  MoveL 6541 to (12.86, -64.22, -148.97) mm, rotated rx 81.04 ry 30.21 rz 20.91 deg; joints [-5.811, -13.888, 75.553, 102.149, 106.889, 54.392, -153.967]
  MoveL 6542 to (13.22, -64.48, -148.9) mm, rotated rx 81.04 ry 30.21 rz 20.91 deg; joints [-5.821, -13.905, 75.562, 102.142, 106.892, 54.402, -153.967]
  MoveL 6543 to (13.58, -64.78, -148.85) mm, rotated rx 81.04 ry 30.21 rz 20.91 deg; joints [-5.832, -13.921, 75.565, 102.137, 106.894, 54.415, -153.967]
  MoveL 6544 to (13.94, -65.11, -148.82) mm, rotated rx 81.04 ry 30.21 rz 20.91 deg; joints [-5.843, -13.936, 75.566, 102.132, 106.896, 54.431, -153.967]
  MoveL 6545 to (14.32, -65.47, -148.8) mm, rotated rx 81.04 ry 30.21 rz 20.91 deg; joints [-5.855, -13.951, 75.564, 102.127, 106.898, 54.45, -153.967]
  MoveL 6546 to (14.69, -65.84, -148.8) mm, rotated rx 81.04 ry 30.21 rz 20.91 deg; joints [-5.866, -13.965, 75.559, 102.123, 106.9, 54.47, -153.967]
  MoveL 6547 to (15.03, -66.17, -148.79) mm, rotated rx 81.04 ry 30.21 rz 20.91 deg; joints [-5.876, -13.978, 75.556, 102.118, 106.901, 54.487, -153.967]
  MoveL 6548 to (15.34, -66.45, -148.76) mm, rotated rx 81.04 ry 30.21 rz 20.91 deg; joints [-5.886, -13.991, 75.556, 102.114, 106.903, 54.501, -153.967]
  MoveL 6549 to (15.69, -66.78, -148.75) mm, rotated rx 81.04 ry 30.21 rz 20.91 deg; joints [-5.897, -14.004, 75.554, 102.11, 106.904, 54.519, -153.967]
  MoveL 6550 to (16.06, -67.16, -148.75) mm, rotated rx 81.04 ry 30.21 rz 20.91 deg; joints [-5.908, -14.018, 75.549, 102.106, 106.906, 54.539, -153.967]
  MoveL 6551 to (16.5, -67.58, -148.73) mm, rotated rx 81.04 ry 30.21 rz 20.91 deg; joints [-5.922, -14.035, 75.546, 102.1, 106.908, 54.561, -153.967]
  MoveL 6552 to (17, -68.06, -148.69) mm, rotated rx 81.04 ry 30.21 rz 20.91 deg; joints [-5.937, -14.056, 75.545, 102.094, 106.91, 54.585, -153.967]
  MoveL 6553 to (17.44, -68.48, -148.67) mm, rotated rx 81.04 ry 30.21 rz 20.91 deg; joints [-5.95, -14.074, 75.542, 102.089, 106.912, 54.607, -153.967]
  MoveL 6554 to (17.9, -68.93, -148.64) mm, rotated rx 81.04 ry 30.21 rz 20.91 deg; joints [-5.964, -14.092, 75.54, 102.083, 106.915, 54.63, -153.967]
  MoveL 6555 to (18.43, -69.41, -148.6) mm, rotated rx 81.04 ry 30.21 rz 20.91 deg; joints [-5.98, -14.113, 75.539, 102.076, 106.917, 54.654, -153.967]
  MoveL 6556 to (18.85, -69.82, -148.59) mm, rotated rx 81.04 ry 30.21 rz 20.91 deg; joints [-5.993, -14.13, 75.535, 102.071, 106.919, 54.676, -153.967]
  MoveL 6557 to (19.24, -70.21, -148.59) mm, rotated rx 81.04 ry 30.21 rz 20.91 deg; joints [-6.005, -14.144, 75.53, 102.066, 106.921, 54.697, -153.967]
  MoveL 6558 to (20.34, -71.32, -148.59) mm, rotated rx 81.04 ry 30.21 rz 20.91 deg; joints [-6.04, -14.184, 75.514, 102.054, 106.925, 54.758, -153.967]
  MoveL 6559 to (21.31, -72.4, -148.67) mm, rotated rx 81.04 ry 30.21 rz 20.91 deg; joints [-6.071, -14.215, 75.486, 102.045, 106.928, 54.822, -153.967]
  MoveL 6560 to (21.99, -73.38, -148.93) mm, rotated rx 81.04 ry 30.21 rz 20.91 deg; joints [-6.094, -14.226, 75.434, 102.044, 106.925, 54.889, -153.967]
  MoveL 6561 to (22.38, -74.25, -149.35) mm, rotated rx 81.04 ry 30.21 rz 20.91 deg; joints [-6.11, -14.216, 75.357, 102.051, 106.919, 54.959, -153.967]
  MoveL 6562 to (22.46, -74.65, -149.62) mm, rotated rx 81.04 ry 30.21 rz 20.91 deg; joints [-6.116, -14.204, 75.309, 102.057, 106.914, 54.996, -153.967]
  MoveL 6563 to (22.47, -75.03, -149.94) mm, rotated rx 81.04 ry 30.21 rz 20.91 deg; joints [-6.119, -14.187, 75.256, 102.064, 106.908, 55.033, -153.967]
  MoveL 6564 to (22.26, -75.71, -150.7) mm, rotated rx 81.04 ry 30.21 rz 20.91 deg; joints [-6.121, -14.137, 75.131, 102.086, 106.893, 55.111, -153.967]
  MoveL 6565 to (21.77, -76.28, -151.62) mm, rotated rx 81.04 ry 30.21 rz 20.91 deg; joints [-6.115, -14.068, 74.981, 102.115, 106.873, 55.192, -153.967]
  MoveL 6566 to (19.9, -77.13, -153.99) mm, rotated rx 81.04 ry 30.21 rz 20.91 deg; joints [-6.08, -13.868, 74.607, 102.195, 106.821, 55.366, -153.967]
  MoveL 6567 to (17.5, -77.39, -156.35) mm, rotated rx 81.04 ry 30.21 rz 20.91 deg; joints [-6.031, -13.647, 74.243, 102.279, 106.766, 55.507, -153.967]
  MoveL 6568 to (15.25, -76.85, -158.04) mm, rotated rx 81.04 ry 30.21 rz 20.91 deg; joints [-5.978, -13.467, 73.999, 102.342, 106.727, 55.567, -153.967]
  MoveL 6569 to (14.17, -76.28, -158.63) mm, rotated rx 81.04 ry 30.21 rz 20.91 deg; joints [-5.951, -13.393, 73.921, 102.365, 106.714, 55.567, -153.967]
  MoveL 6570 to (13.12, -75.52, -159.05) mm, rotated rx 81.04 ry 30.21 rz 20.91 deg; joints [-5.923, -13.329, 73.874, 102.384, 106.704, 55.546, -153.967]
  MoveL 6571 to (11.13, -73.39, -159.39) mm, rotated rx 81.04 ry 30.21 rz 20.91 deg; joints [-5.865, -13.232, 73.871, 102.405, 106.696, 55.444, -153.967]
  MoveL 6572 to (8.58, -70.06, -159.39) mm, rotated rx 81.04 ry 30.21 rz 20.91 deg; joints [-5.787, -13.13, 73.945, 102.419, 106.697, 55.257, -153.967]
  MoveL 6573 to (8.24, -69.63, -159.41) mm, rotated rx 81.04 ry 30.21 rz 20.91 deg; joints [-5.777, -13.115, 73.952, 102.421, 106.697, 55.234, -153.967]
  MoveL 6574 to (7.9, -69.23, -159.45) mm, rotated rx 81.04 ry 30.21 rz 20.91 deg; joints [-5.767, -13.099, 73.955, 102.424, 106.696, 55.213, -153.967]
  MoveL 6575 to (7.54, -68.84, -159.51) mm, rotated rx 81.04 ry 30.21 rz 20.91 deg; joints [-5.757, -13.082, 73.955, 102.428, 106.695, 55.194, -153.967]
  MoveL 6576 to (7.18, -68.47, -159.59) mm, rotated rx 81.04 ry 30.21 rz 20.91 deg; joints [-5.746, -13.062, 73.951, 102.432, 106.693, 55.178, -153.967]
  MoveL 6577 to (6.83, -68.1, -159.67) mm, rotated rx 81.04 ry 30.21 rz 20.91 deg; joints [-5.736, -13.044, 73.947, 102.436, 106.692, 55.161, -153.967]
  MoveL 6578 to (6.52, -67.73, -159.71) mm, rotated rx 81.04 ry 30.21 rz 20.91 deg; joints [-5.727, -13.029, 73.95, 102.439, 106.691, 55.143, -153.967]
  MoveL 6579 to (6.21, -67.35, -159.72) mm, rotated rx 81.04 ry 30.21 rz 20.91 deg; joints [-5.718, -13.016, 73.956, 102.441, 106.691, 55.122, -153.967]
  MoveL 6580 to (5.9, -66.94, -159.72) mm, rotated rx 81.04 ry 30.21 rz 20.91 deg; joints [-5.708, -13.003, 73.965, 102.443, 106.691, 55.099, -153.967]
  MoveL 6581 to (5.5, -66.45, -159.76) mm, rotated rx 81.04 ry 30.21 rz 20.91 deg; joints [-5.697, -12.985, 73.97, 102.446, 106.69, 55.074, -153.967]
  MoveL 6582 to (5.06, -65.93, -159.82) mm, rotated rx 81.04 ry 30.21 rz 20.91 deg; joints [-5.683, -12.964, 73.973, 102.45, 106.689, 55.048, -153.967]
  MoveL 6583 to (4.66, -65.49, -159.84) mm, rotated rx 81.04 ry 30.21 rz 20.91 deg; joints [-5.672, -12.948, 73.979, 102.453, 106.688, 55.024, -153.967]
  MoveL 6584 to (4.27, -65.09, -159.85) mm, rotated rx 81.04 ry 30.21 rz 20.91 deg; joints [-5.659, -12.932, 73.982, 102.458, 106.687, 55.004, -153.967]
  MoveL 6585 to (3.84, -64.74, -159.85) mm, rotated rx 81.04 ry 30.21 rz 20.91 deg; joints [-5.646, -12.917, 73.983, 102.464, 106.684, 54.986, -153.967]
  MoveL 6586 to (3.33, -64.47, -159.85) mm, rotated rx 81.04 ry 30.21 rz 20.91 deg; joints [-5.63, -12.901, 73.977, 102.475, 106.679, 54.974, -153.967]
  MoveL 6587 to (2.76, -64.25, -159.85) mm, rotated rx 81.04 ry 30.21 rz 20.91 deg; joints [-5.612, -12.885, 73.967, 102.488, 106.672, 54.966, -153.967]
  MoveL 6588 to (4.06, -65.14, -160.81) mm, rotated rx 81.04 ry 30.21 rz 20.91 deg; joints [-5.664, -12.861, 73.865, 102.468, 106.679, 55.051, -153.967]
  MoveL 6589 to (2.83, -64.96, -161.23) mm, rotated rx 81.04 ry 30.21 rz 20.91 deg; joints [-5.63, -12.798, 73.778, 102.504, 106.658, 55.071, -153.967]
  MoveL 6590 to (1.45, -64.66, -161.56) mm, rotated rx 81.04 ry 30.21 rz 20.91 deg; joints [-5.59, -12.737, 73.704, 102.541, 106.636, 55.081, -153.967]
  MoveL 6591 to (-0.1, -64.24, -161.81) mm, rotated rx 81.04 ry 30.21 rz 20.91 deg; joints [-5.544, -12.676, 73.637, 102.582, 106.613, 55.081, -153.967]
  MoveL 6592 to (-2.13, -63.57, -161.92) mm, rotated rx 81.04 ry 30.21 rz 20.91 deg; joints [-5.481, -12.609, 73.579, 102.632, 106.585, 55.065, -153.967]
  MoveL 6593 to (-4.16, -62.93, -162.15) mm, rotated rx 81.04 ry 30.21 rz 20.91 deg; joints [-5.42, -12.534, 73.506, 102.683, 106.557, 55.056, -153.967]
  MoveL 6594 to (-6.19, -62.26, -162.26) mm, rotated rx 81.04 ry 30.21 rz 20.91 deg; joints [-5.358, -12.467, 73.447, 102.733, 106.529, 55.041, -153.967]
  MoveL 6595 to (-8.21, -61.59, -162.38) mm, rotated rx 81.04 ry 30.21 rz 20.91 deg; joints [-5.295, -12.399, 73.388, 102.783, 106.501, 55.025, -153.967]
  MoveL 6596 to (-10.24, -60.93, -162.61) mm, rotated rx 81.04 ry 30.21 rz 20.91 deg; joints [-5.234, -12.323, 73.315, 102.834, 106.473, 55.016, -153.967]
  MoveL 6597 to (-12.26, -60.25, -162.73) mm, rotated rx 81.04 ry 30.21 rz 20.91 deg; joints [-5.172, -12.255, 73.255, 102.884, 106.445, 55.001, -153.967]
  MoveL 6598 to (-14.28, -59.57, -162.85) mm, rotated rx 81.04 ry 30.21 rz 20.91 deg; joints [-5.11, -12.187, 73.194, 102.934, 106.418, 54.986, -153.967]
  MoveL 6599 to (-16.62, -58.79, -163.01) mm, rotated rx 81.04 ry 30.21 rz 20.91 deg; joints [-5.038, -12.107, 73.122, 102.992, 106.386, 54.97, -153.967]
  MoveL 6600 to (-18.61, -58.12, -163.21) mm, rotated rx 81.04 ry 30.21 rz 20.91 deg; joints [-4.978, -12.034, 73.054, 103.041, 106.358, 54.958, -153.967]
  MoveL 6601 to (-20.79, -57.37, -163.41) mm, rotated rx 81.04 ry 30.21 rz 20.91 deg; joints [-4.912, -11.955, 72.98, 103.096, 106.328, 54.945, -153.967]
  MoveL 6602 to (-22.93, -56.64, -163.66) mm, rotated rx 81.04 ry 30.21 rz 20.91 deg; joints [-4.848, -11.873, 72.901, 103.149, 106.299, 54.935, -153.967]
  MoveL 6603 to (-24.95, -55.95, -163.78) mm, rotated rx 81.04 ry 30.21 rz 20.91 deg; joints [-4.786, -11.804, 72.839, 103.199, 106.271, 54.92, -153.967]
  MoveL 6604 to (-26.97, -55.26, -163.78) mm, rotated rx 81.04 ry 30.21 rz 20.91 deg; joints [-4.722, -11.743, 72.791, 103.249, 106.244, 54.9, -153.967]
  MoveL 6605 to (-28.96, -54.57, -163.86) mm, rotated rx 81.04 ry 30.21 rz 20.91 deg; joints [-4.661, -11.678, 72.735, 103.298, 106.217, 54.884, -153.967]
  MoveL 6606 to (-30.9, -53.88, -164.07) mm, rotated rx 81.04 ry 30.21 rz 20.91 deg; joints [-4.602, -11.604, 72.665, 103.346, 106.191, 54.873, -153.967]
  MoveL 6607 to (-33.06, -53.09, -164.42) mm, rotated rx 81.04 ry 30.21 rz 20.91 deg; joints [-4.539, -11.513, 72.574, 103.4, 106.161, 54.866, -153.967]
  MoveL 6608 to (-34.75, -52.47, -164.63) mm, rotated rx 81.04 ry 30.21 rz 20.91 deg; joints [-4.488, -11.446, 72.51, 103.442, 106.137, 54.857, -153.967]
  MoveL 6609 to (-37.05, -51.6, -164.93) mm, rotated rx 81.04 ry 30.21 rz 20.91 deg; joints [-4.419, -11.354, 72.423, 103.498, 106.106, 54.844, -153.967]
  MoveL 6610 to (-39.13, -50.86, -165.03) mm, rotated rx 81.04 ry 30.21 rz 20.91 deg; joints [-4.355, -11.283, 72.361, 103.55, 106.078, 54.828, -153.967]
  MoveL 6611 to (-41.15, -50.17, -165.05) mm, rotated rx 81.04 ry 30.21 rz 20.91 deg; joints [-4.292, -11.221, 72.308, 103.6, 106.051, 54.81, -153.967]
  MoveL 6612 to (-41.68, -49.46, -165.84) mm, rotated rx 81.04 ry 30.21 rz 20.91 deg; joints [-4.285, -11.142, 72.231, 103.606, 106.048, 54.808, -153.967]
  MoveL 6613 to (-41.25, -49.43, -166.23) mm, rotated rx 81.04 ry 30.21 rz 20.91 deg; joints [-4.303, -11.126, 72.207, 103.593, 106.054, 54.818, -153.967]
  MoveL 6614 to (-41.11, -49.43, -166.47) mm, rotated rx 81.04 ry 30.21 rz 20.91 deg; joints [-4.31, -11.113, 72.185, 103.589, 106.056, 54.828, -153.967]
  MoveL 6615 to (-41.24, -49.46, -166.6) mm, rotated rx 81.04 ry 30.21 rz 20.91 deg; joints [-4.307, -11.101, 72.163, 103.594, 106.052, 54.837, -153.967]
  MoveL 6616 to (-41.63, -49.55, -166.62) mm, rotated rx 81.04 ry 30.21 rz 20.91 deg; joints [-4.296, -11.09, 72.139, 103.608, 106.044, 54.849, -153.967]
  MoveL 6617 to (-42.08, -49.66, -166.63) mm, rotated rx 81.04 ry 30.21 rz 20.91 deg; joints [-4.281, -11.079, 72.114, 103.624, 106.033, 54.862, -153.967]
  MoveL 6618 to (-43.6, -50.07, -166.63) mm, rotated rx 81.04 ry 30.21 rz 20.91 deg; joints [-4.234, -11.043, 72.028, 103.678, 105.999, 54.907, -153.967]
  MoveL 6619 to (-44.14, -50.2, -166.65) mm, rotated rx 81.04 ry 30.21 rz 20.91 deg; joints [-4.217, -11.029, 71.996, 103.697, 105.987, 54.923, -153.967]
  MoveL 6620 to (-44.68, -50.31, -166.69) mm, rotated rx 81.04 ry 30.21 rz 20.91 deg; joints [-4.201, -11.013, 71.962, 103.716, 105.975, 54.939, -153.967]
  MoveL 6621 to (-45.24, -50.41, -166.77) mm, rotated rx 81.04 ry 30.21 rz 20.91 deg; joints [-4.184, -10.993, 71.923, 103.735, 105.963, 54.956, -153.967]
  MoveL 6622 to (-45.79, -50.51, -166.83) mm, rotated rx 81.04 ry 30.21 rz 20.91 deg; joints [-4.168, -10.976, 71.888, 103.754, 105.951, 54.972, -153.967]
  MoveL 6623 to (-46.3, -50.63, -166.86) mm, rotated rx 81.04 ry 30.21 rz 20.91 deg; joints [-4.152, -10.961, 71.857, 103.772, 105.939, 54.987, -153.967]
  MoveL 6624 to (-46.79, -50.75, -166.88) mm, rotated rx 81.04 ry 30.21 rz 20.91 deg; joints [-4.137, -10.949, 71.828, 103.789, 105.928, 55.002, -153.967]
  MoveL 6625 to (-47.24, -50.84, -166.92) mm, rotated rx 81.04 ry 30.21 rz 20.91 deg; joints [-4.123, -10.934, 71.799, 103.804, 105.918, 55.015, -153.967]
  MoveL 6626 to (-47.67, -50.93, -166.96) mm, rotated rx 81.04 ry 30.21 rz 20.91 deg; joints [-4.11, -10.921, 71.771, 103.819, 105.909, 55.028, -153.967]
  MoveL 6627 to (-48.15, -51.04, -166.98) mm, rotated rx 81.04 ry 30.21 rz 20.91 deg; joints [-4.095, -10.908, 71.743, 103.836, 105.898, 55.042, -153.967]
  MoveL 6628 to (-48.72, -51.18, -167) mm, rotated rx 81.04 ry 30.21 rz 20.91 deg; joints [-4.077, -10.893, 71.709, 103.856, 105.885, 55.059, -153.967]
  MoveL 6629 to (-49.41, -51.32, -167.05) mm, rotated rx 81.04 ry 30.21 rz 20.91 deg; joints [-4.057, -10.873, 71.665, 103.88, 105.87, 55.079, -153.967]
  MoveL 6630 to (-50, -51.46, -167.08) mm, rotated rx 81.04 ry 30.21 rz 20.91 deg; joints [-4.038, -10.857, 71.63, 103.901, 105.856, 55.097, -153.967]
  MoveL 6631 to (-52.03, -52, -167.08) mm, rotated rx 81.04 ry 30.21 rz 20.91 deg; joints [-3.975, -10.808, 71.513, 103.973, 105.81, 55.158, -153.967]
  MoveL 6632 to (-54.91, -52.47, -167.41) mm, rotated rx 81.04 ry 30.21 rz 20.91 deg; joints [-3.889, -10.712, 71.325, 104.07, 105.747, 55.24, -153.967]
  MoveL 6633 to (-56.2, -52.45, -167.82) mm, rotated rx 81.04 ry 30.21 rz 20.91 deg; joints [-3.853, -10.648, 71.222, 104.111, 105.72, 55.275, -153.967]
  MoveL 6634 to (-57.4, -52.25, -168.4) mm, rotated rx 81.04 ry 30.21 rz 20.91 deg; joints [-3.823, -10.572, 71.112, 104.145, 105.698, 55.305, -153.967]
  MoveL 6635 to (-59.51, -51.31, -170.05) mm, rotated rx 81.04 ry 30.21 rz 20.91 deg; joints [-3.777, -10.386, 70.875, 104.198, 105.663, 55.351, -153.967]
  MoveL 6636 to (-61.23, -49.68, -172.36) mm, rotated rx 81.04 ry 30.21 rz 20.91 deg; joints [-3.75, -10.156, 70.613, 104.229, 105.642, 55.38, -153.967]
  MoveL 6637 to (-62.18, -47.89, -174.66) mm, rotated rx 81.04 ry 30.21 rz 20.91 deg; joints [-3.748, -9.944, 70.391, 104.233, 105.639, 55.39, -153.967]
  MoveL 6638 to (-62.22, -47.14, -175.57) mm, rotated rx 81.04 ry 30.21 rz 20.91 deg; joints [-3.758, -9.87, 70.322, 104.224, 105.645, 55.386, -153.967]
  MoveL 6639 to (-61.96, -46.49, -176.31) mm, rotated rx 81.04 ry 30.21 rz 20.91 deg; joints [-3.775, -9.816, 70.279, 104.207, 105.656, 55.377, -153.967]
  MoveL 6640 to (-61.72, -46.2, -176.62) mm, rotated rx 81.04 ry 30.21 rz 20.91 deg; joints [-3.786, -9.797, 70.268, 104.195, 105.663, 55.37, -153.967]
  MoveL 6641 to (-61.41, -45.94, -176.89) mm, rotated rx 81.04 ry 30.21 rz 20.91 deg; joints [-3.799, -9.784, 70.264, 104.182, 105.671, 55.362, -153.967]
  MoveL 6642 to (-60.57, -45.48, -177.3) mm, rotated rx 81.04 ry 30.21 rz 20.91 deg; joints [-3.83, -9.772, 70.277, 104.149, 105.692, 55.342, -153.967]
  MoveL 6643 to (-59.44, -45.12, -177.55) mm, rotated rx 81.04 ry 30.21 rz 20.91 deg; joints [-3.868, -9.781, 70.317, 104.109, 105.718, 55.315, -153.967]
  MoveL 6644 to (-58.01, -44.86, -177.63) mm, rotated rx 81.04 ry 30.21 rz 20.91 deg; joints [-3.914, -9.811, 70.384, 104.06, 105.749, 55.283, -153.967]
  MoveL 6645 to (-54.38, -44.37, -177.63) mm, rotated rx 81.04 ry 30.21 rz 20.91 deg; joints [-4.027, -9.905, 70.571, 103.94, 105.825, 55.203, -153.967]
  MoveL 6646 to (-53.92, -44.32, -177.61) mm, rotated rx 81.04 ry 30.21 rz 20.91 deg; joints [-4.041, -9.918, 70.596, 103.925, 105.835, 55.193, -153.967]
  MoveL 6647 to (-53.51, -44.29, -177.59) mm, rotated rx 81.04 ry 30.21 rz 20.91 deg; joints [-4.054, -9.93, 70.619, 103.911, 105.843, 55.184, -153.967]
  MoveL 6648 to (-53.04, -44.23, -177.57) mm, rotated rx 81.04 ry 30.21 rz 20.91 deg; joints [-4.068, -9.944, 70.645, 103.896, 105.853, 55.174, -153.967]
  MoveL 6649 to (-49.4, -43.75, -177.57) mm, rotated rx 81.04 ry 30.21 rz 20.91 deg; joints [-4.182, -10.036, 70.829, 103.775, 105.929, 55.094, -153.967]
  MoveL 6650 to (-48.86, -43.7, -177.55) mm, rotated rx 81.04 ry 30.21 rz 20.91 deg; joints [-4.199, -10.052, 70.858, 103.757, 105.94, 55.083, -153.967]
  MoveL 6651 to (-48.32, -43.68, -177.51) mm, rotated rx 81.04 ry 30.21 rz 20.91 deg; joints [-4.215, -10.069, 70.887, 103.74, 105.951, 55.073, -153.967]
  MoveL 6652 to (-47.83, -43.71, -177.47) mm, rotated rx 81.04 ry 30.21 rz 20.91 deg; joints [-4.23, -10.086, 70.912, 103.725, 105.96, 55.066, -153.967]
  MoveL 6653 to (-47.45, -43.76, -177.41) mm, rotated rx 81.04 ry 30.21 rz 20.91 deg; joints [-4.241, -10.101, 70.933, 103.714, 105.966, 55.062, -153.967]
  MoveL 6654 to (-47.27, -43.83, -177.24) mm, rotated rx 81.04 ry 30.21 rz 20.91 deg; joints [-4.245, -10.118, 70.957, 103.709, 105.97, 55.056, -153.967]
  MoveL 6655 to (-47.26, -43.87, -176.91) mm, rotated rx 81.04 ry 30.21 rz 20.91 deg; joints [-4.241, -10.142, 70.994, 103.709, 105.971, 55.042, -153.967]
  MoveL 6656 to (-47.42, -43.87, -176.4) mm, rotated rx 81.04 ry 30.21 rz 20.91 deg; joints [-4.23, -10.175, 71.046, 103.712, 105.971, 55.021, -153.967]
  MoveL 6657 to (-47.11, -44.64, -174.94) mm, rotated rx 81.04 ry 30.21 rz 20.91 deg; joints [-4.223, -10.296, 71.191, 103.712, 105.973, 54.996, -153.967]
  MoveL 6658 to (-43.28, -46.52, -174.94) mm, rotated rx 81.04 ry 30.21 rz 20.91 deg; joints [-4.342, -10.421, 71.262, 103.627, 106.017, 55.065, -153.967]
  MoveL 6659 to (-41.45, -47.43, -174.89) mm, rotated rx 81.04 ry 30.21 rz 20.91 deg; joints [-4.399, -10.484, 71.301, 103.586, 106.038, 55.096, -153.967]
  MoveL 6660 to (-39.68, -48.31, -174.8) mm, rotated rx 81.04 ry 30.21 rz 20.91 deg; joints [-4.453, -10.547, 71.343, 103.546, 106.058, 55.124, -153.967]
  MoveL 6661 to (-37.88, -49.2, -174.72) mm, rotated rx 81.04 ry 30.21 rz 20.91 deg; joints [-4.509, -10.612, 71.385, 103.506, 106.079, 55.154, -153.967]
  MoveL 6662 to (-36.11, -50.07, -174.62) mm, rotated rx 81.04 ry 30.21 rz 20.91 deg; joints [-4.562, -10.676, 71.428, 103.467, 106.1, 55.182, -153.967]
  MoveL 6663 to (-34.24, -51.02, -174.58) mm, rotated rx 81.04 ry 30.21 rz 20.91 deg; joints [-4.62, -10.739, 71.463, 103.426, 106.121, 55.216, -153.967]
  MoveL 6664 to (-32.32, -52.09, -174.54) mm, rotated rx 81.04 ry 30.21 rz 20.91 deg; joints [-4.68, -10.805, 71.495, 103.386, 106.142, 55.258, -153.967]
  MoveL 6665 to (-30.03, -53.11, -174.38) mm, rotated rx 81.04 ry 30.21 rz 20.91 deg; joints [-4.749, -10.889, 71.559, 103.333, 106.17, 55.287, -153.967]
  MoveL 6666 to (-28.02, -54.1, -174.13) mm, rotated rx 81.04 ry 30.21 rz 20.91 deg; joints [-4.809, -10.971, 71.622, 103.288, 106.194, 55.313, -153.967]
  MoveL 6667 to (-26.05, -55.07, -174) mm, rotated rx 81.04 ry 30.21 rz 20.91 deg; joints [-4.869, -11.043, 71.67, 103.245, 106.217, 55.345, -153.967]
  MoveL 6668 to (-24.14, -56, -173.76) mm, rotated rx 81.04 ry 30.21 rz 20.91 deg; joints [-4.926, -11.121, 71.73, 103.202, 106.24, 55.37, -153.967]
  MoveL 6669 to (-22.22, -56.94, -173.64) mm, rotated rx 81.04 ry 30.21 rz 20.91 deg; joints [-4.985, -11.191, 71.775, 103.16, 106.263, 55.401, -153.967]
  MoveL 6670 to (-20.3, -57.87, -173.52) mm, rotated rx 81.04 ry 30.21 rz 20.91 deg; joints [-5.043, -11.26, 71.82, 103.117, 106.285, 55.432, -153.967]
  MoveL 6671 to (-18.38, -58.8, -173.28) mm, rotated rx 81.04 ry 30.21 rz 20.91 deg; joints [-5.101, -11.337, 71.88, 103.074, 106.309, 55.456, -153.967]
  MoveL 6672 to (-16.45, -59.72, -173.16) mm, rotated rx 81.04 ry 30.21 rz 20.91 deg; joints [-5.159, -11.406, 71.925, 103.032, 106.332, 55.487, -153.967]
  MoveL 6673 to (-14.53, -60.65, -173.04) mm, rotated rx 81.04 ry 30.21 rz 20.91 deg; joints [-5.218, -11.475, 71.969, 102.99, 106.354, 55.519, -153.967]
  MoveL 6674 to (-12.61, -61.57, -172.92) mm, rotated rx 81.04 ry 30.21 rz 20.91 deg; joints [-5.276, -11.543, 72.014, 102.948, 106.377, 55.55, -153.967]
  MoveL 6675 to (-10.68, -62.48, -172.69) mm, rotated rx 81.04 ry 30.21 rz 20.91 deg; joints [-5.334, -11.619, 72.072, 102.905, 106.401, 55.575, -153.967]
  MoveL 6676 to (-8.75, -63.4, -172.58) mm, rotated rx 81.04 ry 30.21 rz 20.91 deg; joints [-5.393, -11.687, 72.115, 102.862, 106.423, 55.607, -153.967]
  MoveL 6677 to (-7.12, -64.13, -172.33) mm, rotated rx 81.04 ry 30.21 rz 20.91 deg; joints [-5.441, -11.755, 72.171, 102.825, 106.444, 55.624, -153.967]
  MoveL 6678 to (-5.6, -64.79, -172.01) mm, rotated rx 81.04 ry 30.21 rz 20.91 deg; joints [-5.485, -11.824, 72.235, 102.79, 106.464, 55.634, -153.967]
  MoveL 6679 to (-4.15, -65.39, -171.59) mm, rotated rx 81.04 ry 30.21 rz 20.91 deg; joints [-5.525, -11.897, 72.31, 102.756, 106.484, 55.638, -153.967]
  MoveL 6680 to (-5.26, -64.05, -170.63) mm, rotated rx 81.04 ry 30.21 rz 20.91 deg; joints [-5.48, -11.922, 72.444, 102.762, 106.486, 55.521, -153.967]
  MoveL 6681 to (-4.71, -64.37, -170.51) mm, rotated rx 81.04 ry 30.21 rz 20.91 deg; joints [-5.496, -11.948, 72.464, 102.751, 106.492, 55.529, -153.967]
  MoveL 6682 to (-4.24, -64.71, -170.42) mm, rotated rx 81.04 ry 30.21 rz 20.91 deg; joints [-5.51, -11.97, 72.475, 102.743, 106.496, 55.542, -153.967]
  MoveL 6683 to (-3.88, -65.12, -170.39) mm, rotated rx 81.04 ry 30.21 rz 20.91 deg; joints [-5.521, -11.987, 72.472, 102.739, 106.498, 55.563, -153.967]
  MoveL 6684 to (-3.56, -65.54, -170.37) mm, rotated rx 81.04 ry 30.21 rz 20.91 deg; joints [-5.53, -12.001, 72.465, 102.737, 106.497, 55.586, -153.967]
  MoveL 6685 to (-1.7, -68.72, -170.36) mm, rotated rx 81.04 ry 30.21 rz 20.91 deg; joints [-5.587, -12.084, 72.375, 102.74, 106.487, 55.767, -153.967]
  MoveL 6686 to (-1.46, -69.11, -170.35) mm, rotated rx 81.04 ry 30.21 rz 20.91 deg; joints [-5.594, -12.095, 72.366, 102.74, 106.485, 55.79, -153.967]
  MoveL 6687 to (-1.23, -69.47, -170.32) mm, rotated rx 81.04 ry 30.21 rz 20.91 deg; joints [-5.6, -12.107, 72.359, 102.739, 106.485, 55.809, -153.967]
  MoveL 6688 to (-0.99, -69.88, -170.31) mm, rotated rx 81.04 ry 30.21 rz 20.91 deg; joints [-5.608, -12.118, 72.349, 102.74, 106.483, 55.832, -153.967]
  MoveL 6689 to (-0.72, -70.34, -170.31) mm, rotated rx 81.04 ry 30.21 rz 20.91 deg; joints [-5.616, -12.13, 72.336, 102.74, 106.482, 55.858, -153.967]
  MoveL 6690 to (0.06, -71.7, -170.31) mm, rotated rx 81.04 ry 30.21 rz 20.91 deg; joints [-5.639, -12.165, 72.296, 102.742, 106.477, 55.937, -153.967]
  MoveL 6691 to (0.39, -72.23, -170.29) mm, rotated rx 81.04 ry 30.21 rz 20.91 deg; joints [-5.649, -12.18, 72.283, 102.742, 106.475, 55.967, -153.967]
  MoveL 6692 to (0.77, -72.84, -170.25) mm, rotated rx 81.04 ry 30.21 rz 20.91 deg; joints [-5.66, -12.199, 72.271, 102.741, 106.474, 56, -153.967]
  MoveL 6693 to (1.11, -73.39, -170.23) mm, rotated rx 81.04 ry 30.21 rz 20.91 deg; joints [-5.67, -12.215, 72.258, 102.742, 106.472, 56.03, -153.967]
  MoveL 6694 to (1.63, -74.29, -170.23) mm, rotated rx 81.04 ry 30.21 rz 20.91 deg; joints [-5.686, -12.238, 72.231, 102.743, 106.469, 56.083, -153.967]
  MoveL 6695 to (2.29, -75.58, -170.32) mm, rotated rx 81.04 ry 30.21 rz 20.91 deg; joints [-5.707, -12.262, 72.18, 102.747, 106.463, 56.162, -153.967]
  MoveL 6696 to (2.7, -76.7, -170.57) mm, rotated rx 81.04 ry 30.21 rz 20.91 deg; joints [-5.722, -12.266, 72.108, 102.757, 106.453, 56.241, -153.967]
  MoveL 6697 to (2.84, -77.64, -170.99) mm, rotated rx 81.04 ry 30.21 rz 20.91 deg; joints [-5.73, -12.25, 72.016, 102.771, 106.44, 56.319, -153.967]
  MoveL 6698 to (2.82, -78.04, -171.26) mm, rotated rx 81.04 ry 30.21 rz 20.91 deg; joints [-5.732, -12.234, 71.962, 102.781, 106.433, 56.358, -153.967]
  MoveL 6699 to (2.73, -78.41, -171.58) mm, rotated rx 81.04 ry 30.21 rz 20.91 deg; joints [-5.733, -12.213, 71.903, 102.791, 106.425, 56.396, -153.967]
  MoveL 6700 to (2.35, -79, -172.33) mm, rotated rx 81.04 ry 30.21 rz 20.91 deg; joints [-5.729, -12.156, 71.77, 102.816, 106.406, 56.473, -153.967]
  MoveL 6701 to (1.72, -79.42, -173.26) mm, rotated rx 81.04 ry 30.21 rz 20.91 deg; joints [-5.719, -12.078, 71.616, 102.846, 106.384, 56.549, -153.967]
  MoveL 6702 to (-0.33, -79.75, -175.61) mm, rotated rx 81.04 ry 30.21 rz 20.91 deg; joints [-5.681, -11.86, 71.245, 102.922, 106.331, 56.7, -153.967]
  MoveL 6703 to (-2.73, -79.36, -177.96) mm, rotated rx 81.04 ry 30.21 rz 20.91 deg; joints [-5.632, -11.625, 70.896, 102.994, 106.282, 56.81, -153.967]
  MoveL 6704 to (-4.79, -78.25, -179.64) mm, rotated rx 81.04 ry 30.21 rz 20.91 deg; joints [-5.587, -11.439, 70.676, 103.041, 106.252, 56.839, -153.967]
  MoveL 6705 to (-5.69, -77.42, -180.23) mm, rotated rx 81.04 ry 30.21 rz 20.91 deg; joints [-5.566, -11.365, 70.615, 103.055, 106.244, 56.823, -153.967]
  MoveL 6706 to (-6.51, -76.41, -180.65) mm, rotated rx 81.04 ry 30.21 rz 20.91 deg; joints [-5.546, -11.304, 70.587, 103.062, 106.241, 56.787, -153.967]
  MoveL 6707 to (-7.9, -73.84, -180.98) mm, rotated rx 81.04 ry 30.21 rz 20.91 deg; joints [-5.508, -11.218, 70.628, 103.058, 106.251, 56.654, -153.967]
  MoveL 6708 to (-9.11, -70.94, -180.98) mm, rotated rx 81.04 ry 30.21 rz 20.91 deg; joints [-5.472, -11.158, 70.733, 103.041, 106.271, 56.482, -153.967]
  MoveL 6709 to (-9.53, -70.05, -181.03) mm, rotated rx 81.04 ry 30.21 rz 20.91 deg; joints [-5.46, -11.134, 70.757, 103.037, 106.275, 56.432, -153.967]
  MoveL 6710 to (-9.73, -69.57, -181.03) mm, rotated rx 81.04 ry 30.21 rz 20.91 deg; joints [-5.454, -11.124, 70.774, 103.034, 106.279, 56.404, -153.967]
  MoveL 6711 to (-9.94, -69.07, -181.03) mm, rotated rx 81.04 ry 30.21 rz 20.91 deg; joints [-5.447, -11.113, 70.791, 103.031, 106.282, 56.374, -153.967]
  MoveL 6712 to (-10.17, -68.55, -181.06) mm, rotated rx 81.04 ry 30.21 rz 20.91 deg; joints [-5.441, -11.1, 70.807, 103.029, 106.285, 56.345, -153.967]
  MoveL 6713 to (-10.46, -67.97, -181.12) mm, rotated rx 81.04 ry 30.21 rz 20.91 deg; joints [-5.433, -11.082, 70.819, 103.027, 106.288, 56.314, -153.967]
  MoveL 6714 to (-10.7, -67.44, -181.15) mm, rotated rx 81.04 ry 30.21 rz 20.91 deg; joints [-5.426, -11.068, 70.833, 103.025, 106.291, 56.284, -153.967]
  MoveL 6715 to (-10.91, -66.96, -181.16) mm, rotated rx 81.04 ry 30.21 rz 20.91 deg; joints [-5.42, -11.057, 70.848, 103.022, 106.294, 56.257, -153.967]
  MoveL 6716 to (-11.11, -66.53, -181.19) mm, rotated rx 81.04 ry 30.21 rz 20.91 deg; joints [-5.414, -11.045, 70.859, 103.021, 106.296, 56.233, -153.967]
  MoveL 6717 to (-11.32, -66.13, -181.24) mm, rotated rx 81.04 ry 30.21 rz 20.91 deg; joints [-5.408, -11.032, 70.866, 103.02, 106.298, 56.212, -153.967]
  MoveL 6718 to (-11.52, -65.71, -181.28) mm, rotated rx 81.04 ry 30.21 rz 20.91 deg; joints [-5.403, -11.019, 70.875, 103.018, 106.3, 56.19, -153.967]
  MoveL 6719 to (-11.73, -65.25, -181.29) mm, rotated rx 81.04 ry 30.21 rz 20.91 deg; joints [-5.397, -11.008, 70.889, 103.016, 106.303, 56.163, -153.967]
  MoveL 6720 to (-11.94, -64.78, -181.3) mm, rotated rx 81.04 ry 30.21 rz 20.91 deg; joints [-5.39, -10.998, 70.904, 103.014, 106.306, 56.136, -153.967]
  MoveL 6721 to (-12.17, -64.32, -181.3) mm, rotated rx 81.04 ry 30.21 rz 20.91 deg; joints [-5.384, -10.986, 70.918, 103.012, 106.308, 56.109, -153.967]
  MoveL 6722 to (-12.43, -63.91, -181.32) mm, rotated rx 81.04 ry 30.21 rz 20.91 deg; joints [-5.376, -10.973, 70.927, 103.013, 106.309, 56.087, -153.967]
  MoveL 6723 to (-12.74, -63.54, -181.35) mm, rotated rx 81.04 ry 30.21 rz 20.91 deg; joints [-5.367, -10.959, 70.93, 103.015, 106.308, 56.069, -153.967]
  MoveL 6724 to (-13.08, -63.24, -181.4) mm, rotated rx 81.04 ry 30.21 rz 20.91 deg; joints [-5.357, -10.944, 70.926, 103.02, 106.306, 56.055, -153.967]
  MoveL 6725 to (-13.44, -62.96, -181.44) mm, rotated rx 81.04 ry 30.21 rz 20.91 deg; joints [-5.346, -10.928, 70.921, 103.026, 106.303, 56.044, -153.967]
  MoveL 6726 to (-12.41, -64.08, -182.41) mm, rotated rx 81.04 ry 30.21 rz 20.91 deg; joints [-5.389, -10.898, 70.791, 103.019, 106.302, 56.149, -153.967]
  MoveL 6727 to (-13.93, -63.28, -182.79) mm, rotated rx 81.04 ry 30.21 rz 20.91 deg; joints [-5.346, -10.822, 70.726, 103.052, 106.283, 56.133, -153.967]
  MoveL 6728 to (-15.5, -62.38, -183.07) mm, rotated rx 81.04 ry 30.21 rz 20.91 deg; joints [-5.3, -10.752, 70.676, 103.084, 106.265, 56.108, -153.967]
  MoveL 6729 to (-17.16, -61.37, -183.27) mm, rotated rx 81.04 ry 30.21 rz 20.91 deg; joints [-5.251, -10.683, 70.636, 103.117, 106.248, 56.072, -153.967]
  MoveL 6730 to (-18.97, -60.23, -183.49) mm, rotated rx 81.04 ry 30.21 rz 20.91 deg; joints [-5.197, -10.607, 70.594, 103.152, 106.229, 56.032, -153.967]
  MoveL 6731 to (-20.76, -59.07, -183.61) mm, rotated rx 81.04 ry 30.21 rz 20.91 deg; joints [-5.143, -10.539, 70.566, 103.185, 106.212, 55.985, -153.967]
  MoveL 6732 to (-22.55, -57.91, -183.72) mm, rotated rx 81.04 ry 30.21 rz 20.91 deg; joints [-5.089, -10.472, 70.538, 103.219, 106.195, 55.938, -153.967]
  MoveL 6733 to (-24.35, -56.75, -183.95) mm, rotated rx 81.04 ry 30.21 rz 20.91 deg; joints [-5.036, -10.395, 70.494, 103.254, 106.177, 55.898, -153.967]
  MoveL 6734 to (-26.14, -55.59, -184.07) mm, rotated rx 81.04 ry 30.21 rz 20.91 deg; joints [-4.982, -10.326, 70.465, 103.288, 106.16, 55.852, -153.967]
  MoveL 6735 to (-27.92, -54.42, -184.19) mm, rotated rx 81.04 ry 30.21 rz 20.91 deg; joints [-4.928, -10.258, 70.436, 103.322, 106.143, 55.805, -153.967]
  MoveL 6736 to (-29.71, -53.25, -184.43) mm, rotated rx 81.04 ry 30.21 rz 20.91 deg; joints [-4.875, -10.18, 70.392, 103.357, 106.125, 55.765, -153.967]
  MoveL 6737 to (-31.49, -52.08, -184.55) mm, rotated rx 81.04 ry 30.21 rz 20.91 deg; joints [-4.821, -10.111, 70.362, 103.391, 106.108, 55.719, -153.967]
  MoveL 6738 to (-33.27, -50.9, -184.67) mm, rotated rx 81.04 ry 30.21 rz 20.91 deg; joints [-4.767, -10.042, 70.332, 103.425, 106.091, 55.673, -153.967]
  MoveL 6739 to (-34.95, -49.78, -184.86) mm, rotated rx 81.04 ry 30.21 rz 20.91 deg; joints [-4.718, -9.971, 70.295, 103.457, 106.075, 55.633, -153.967]
  MoveL 6740 to (-36.47, -48.77, -185.07) mm, rotated rx 81.04 ry 30.21 rz 20.91 deg; joints [-4.673, -9.903, 70.256, 103.486, 106.06, 55.599, -153.967]
  MoveL 6741 to (-38.1, -47.68, -185.18) mm, rotated rx 81.04 ry 30.21 rz 20.91 deg; joints [-4.623, -9.84, 70.229, 103.517, 106.044, 55.556, -153.967]
  MoveL 6742 to (-39.97, -46.56, -185.18) mm, rotated rx 81.04 ry 30.21 rz 20.91 deg; joints [-4.565, -9.777, 70.205, 103.555, 106.026, 55.51, -153.967]
  MoveL 6743 to (-42.22, -45.04, -185.27) mm, rotated rx 81.04 ry 30.21 rz 20.91 deg; joints [-4.496, -9.693, 70.173, 103.598, 106.005, 55.448, -153.967]
  MoveL 6744 to (-44.2, -43.57, -185.51) mm, rotated rx 81.04 ry 30.21 rz 20.91 deg; joints [-4.438, -9.605, 70.133, 103.634, 105.988, 55.393, -153.967]
  MoveL 6745 to (-45.88, -42.42, -185.69) mm, rotated rx 81.04 ry 30.21 rz 20.91 deg; joints [-4.387, -9.534, 70.096, 103.667, 105.972, 55.353, -153.967]
  MoveL 6746 to (-47.42, -41.36, -186.01) mm, rotated rx 81.04 ry 30.21 rz 20.91 deg; joints [-4.343, -9.457, 70.044, 103.697, 105.957, 55.322, -153.967]
  MoveL 6747 to (-49.11, -40.2, -186.19) mm, rotated rx 81.04 ry 30.21 rz 20.91 deg; joints [-4.293, -9.385, 70.006, 103.729, 105.941, 55.281, -153.967]
  MoveL 6748 to (-50.72, -39.07, -186.39) mm, rotated rx 81.04 ry 30.21 rz 20.91 deg; joints [-4.245, -9.313, 69.968, 103.76, 105.926, 55.242, -153.967]
  MoveL 6749 to (-52.29, -37.94, -186.67) mm, rotated rx 81.04 ry 30.21 rz 20.91 deg; joints [-4.2, -9.237, 69.921, 103.79, 105.912, 55.206, -153.967]
  MoveL 6750 to (-52.59, -37.09, -187.44) mm, rotated rx 81.04 ry 30.21 rz 20.91 deg; joints [-4.199, -9.164, 69.86, 103.787, 105.914, 55.194, -153.967]
  MoveL 6751 to (-52.22, -37.11, -187.82) mm, rotated rx 81.04 ry 30.21 rz 20.91 deg; joints [-4.216, -9.146, 69.83, 103.777, 105.919, 55.209, -153.967]
  MoveL 6752 to (-52.14, -37.09, -188.06) mm, rotated rx 81.04 ry 30.21 rz 20.91 deg; joints [-4.221, -9.131, 69.806, 103.775, 105.92, 55.218, -153.967]
  MoveL 6753 to (-52.34, -37.03, -188.19) mm, rotated rx 81.04 ry 30.21 rz 20.91 deg; joints [-4.216, -9.115, 69.785, 103.781, 105.916, 55.224, -153.967]
  MoveL 6754 to (-52.86, -36.97, -188.24) mm, rotated rx 81.04 ry 30.21 rz 20.91 deg; joints [-4.2, -9.097, 69.758, 103.796, 105.907, 55.23, -153.967]
  MoveL 6755 to (-53.53, -36.93, -188.28) mm, rotated rx 81.04 ry 30.21 rz 20.91 deg; joints [-4.18, -9.076, 69.726, 103.816, 105.894, 55.238, -153.967]
  MoveL 6756 to (-55.1, -36.94, -188.28) mm, rotated rx 81.04 ry 30.21 rz 20.91 deg; joints [-4.131, -9.033, 69.655, 103.865, 105.864, 55.26, -153.967]
  MoveL 6757 to (-55.65, -36.94, -188.28) mm, rotated rx 81.04 ry 30.21 rz 20.91 deg; joints [-4.114, -9.017, 69.63, 103.882, 105.854, 55.268, -153.967]
  MoveL 6758 to (-56.18, -36.92, -188.31) mm, rotated rx 81.04 ry 30.21 rz 20.91 deg; joints [-4.098, -9.001, 69.604, 103.898, 105.844, 55.276, -153.967]
  MoveL 6759 to (-56.73, -36.89, -188.36) mm, rotated rx 81.04 ry 30.21 rz 20.91 deg; joints [-4.081, -8.982, 69.575, 103.915, 105.833, 55.284, -153.967]
  MoveL 6760 to (-57.29, -36.84, -188.43) mm, rotated rx 81.04 ry 30.21 rz 20.91 deg; joints [-4.065, -8.961, 69.543, 103.931, 105.823, 55.292, -153.967]
  MoveL 6761 to (-57.84, -36.8, -188.49) mm, rotated rx 81.04 ry 30.21 rz 20.91 deg; joints [-4.048, -8.941, 69.513, 103.948, 105.813, 55.301, -153.967]
  MoveL 6762 to (-58.34, -36.79, -188.51) mm, rotated rx 81.04 ry 30.21 rz 20.91 deg; joints [-4.033, -8.925, 69.489, 103.963, 105.803, 55.308, -153.967]
  MoveL 6763 to (-58.79, -36.78, -188.53) mm, rotated rx 81.04 ry 30.21 rz 20.91 deg; joints [-4.019, -8.912, 69.467, 103.977, 105.795, 55.315, -153.967]
  MoveL 6764 to (-60.36, -36.79, -188.53) mm, rotated rx 81.04 ry 30.21 rz 20.91 deg; joints [-3.97, -8.868, 69.395, 104.026, 105.764, 55.337, -153.967]
  MoveL 6765 to (-60.88, -36.78, -188.54) mm, rotated rx 81.04 ry 30.21 rz 20.91 deg; joints [-3.954, -8.853, 69.37, 104.042, 105.754, 55.345, -153.967]
  MoveL 6766 to (-61.36, -36.76, -188.57) mm, rotated rx 81.04 ry 30.21 rz 20.91 deg; joints [-3.939, -8.838, 69.346, 104.056, 105.745, 55.352, -153.967]
  MoveL 6767 to (-61.8, -36.73, -188.62) mm, rotated rx 81.04 ry 30.21 rz 20.91 deg; joints [-3.926, -8.821, 69.322, 104.07, 105.737, 55.358, -153.967]
  MoveL 6768 to (-62.26, -36.7, -188.66) mm, rotated rx 81.04 ry 30.21 rz 20.91 deg; joints [-3.912, -8.806, 69.298, 104.084, 105.728, 55.365, -153.967]
  MoveL 6769 to (-62.75, -36.69, -188.67) mm, rotated rx 81.04 ry 30.21 rz 20.91 deg; joints [-3.897, -8.791, 69.274, 104.099, 105.719, 55.372, -153.967]
  MoveL 6770 to (-63.27, -36.69, -188.67) mm, rotated rx 81.04 ry 30.21 rz 20.91 deg; joints [-3.881, -8.777, 69.25, 104.115, 105.709, 55.38, -153.967]
  MoveL 6771 to (-66.19, -36.41, -189.01) mm, rotated rx 81.04 ry 30.21 rz 20.91 deg; joints [-3.794, -8.668, 69.09, 104.201, 105.655, 55.421, -153.967]
  MoveL 6772 to (-67.45, -36.05, -189.43) mm, rotated rx 81.04 ry 30.21 rz 20.91 deg; joints [-3.76, -8.598, 68.999, 104.236, 105.633, 55.437, -153.967]
  MoveL 6773 to (-68.59, -35.54, -190.02) mm, rotated rx 81.04 ry 30.21 rz 20.91 deg; joints [-3.732, -8.518, 68.902, 104.264, 105.616, 55.451, -153.967]
  MoveL 6774 to (-70.47, -34.08, -191.71) mm, rotated rx 81.04 ry 30.21 rz 20.91 deg; joints [-3.693, -8.326, 68.684, 104.303, 105.591, 55.472, -153.967]
  MoveL 6775 to (-71.84, -32.03, -194.07) mm, rotated rx 81.04 ry 30.21 rz 20.91 deg; joints [-3.679, -8.091, 68.438, 104.318, 105.581, 55.482, -153.967]
  MoveL 6776 to (-72.42, -30.03, -196.43) mm, rotated rx 81.04 ry 30.21 rz 20.91 deg; joints [-3.689, -7.879, 68.224, 104.31, 105.586, 55.485, -153.967]
  MoveL 6777 to (-72.31, -29.28, -197.36) mm, rotated rx 81.04 ry 30.21 rz 20.91 deg; joints [-3.703, -7.806, 68.154, 104.297, 105.593, 55.483, -153.967]
  MoveL 6778 to (-71.93, -28.71, -198.12) mm, rotated rx 81.04 ry 30.21 rz 20.91 deg; joints [-3.724, -7.754, 68.108, 104.278, 105.605, 55.48, -153.967]
  MoveL 6779 to (-71.64, -28.49, -198.44) mm, rotated rx 81.04 ry 30.21 rz 20.91 deg; joints [-3.737, -7.736, 68.094, 104.267, 105.612, 55.478, -153.967]
  MoveL 6780 to (-71.29, -28.31, -198.71) mm, rotated rx 81.04 ry 30.21 rz 20.91 deg; joints [-3.751, -7.724, 68.086, 104.254, 105.619, 55.476, -153.967]
  MoveL 6781 to (-70.38, -28.07, -199.13) mm, rotated rx 81.04 ry 30.21 rz 20.91 deg; joints [-3.784, -7.716, 68.089, 104.223, 105.638, 55.469, -153.967]
  MoveL 6782 to (-69.2, -28.01, -199.39) mm, rotated rx 81.04 ry 30.21 rz 20.91 deg; joints [-3.824, -7.73, 68.116, 104.186, 105.66, 55.46, -153.967]
  MoveL 6783 to (-67.76, -28.12, -199.47) mm, rotated rx 81.04 ry 30.21 rz 20.91 deg; joints [-3.87, -7.765, 68.167, 104.144, 105.686, 55.45, -153.967]
  MoveL 6784 to (-66.2, -28.32, -199.47) mm, rotated rx 81.04 ry 30.21 rz 20.91 deg; joints [-3.918, -7.811, 68.23, 104.099, 105.714, 55.439, -153.967]
  MoveL 6785 to (-65.68, -28.39, -199.47) mm, rotated rx 81.04 ry 30.21 rz 20.91 deg; joints [-3.934, -7.827, 68.252, 104.084, 105.723, 55.435, -153.967]
  MoveL 6786 to (-65.11, -28.48, -199.43) mm, rotated rx 81.04 ry 30.21 rz 20.91 deg; joints [-3.952, -7.846, 68.277, 104.067, 105.732, 55.431, -153.967]
  MoveL 6787 to (-64.48, -28.61, -199.37) mm, rotated rx 81.04 ry 30.21 rz 20.91 deg; joints [-3.97, -7.87, 68.308, 104.05, 105.743, 55.426, -153.967]
  MoveL 6788 to (-63.92, -28.7, -199.34) mm, rotated rx 81.04 ry 30.21 rz 20.91 deg; joints [-3.987, -7.889, 68.333, 104.034, 105.753, 55.422, -153.967]
  MoveL 6789 to (-63.39, -28.77, -199.34) mm, rotated rx 81.04 ry 30.21 rz 20.91 deg; joints [-4.004, -7.904, 68.354, 104.019, 105.762, 55.419, -153.967]
  MoveL 6790 to (-62.88, -28.84, -199.33) mm, rotated rx 81.04 ry 30.21 rz 20.91 deg; joints [-4.02, -7.92, 68.376, 104.004, 105.771, 55.415, -153.967]
  MoveL 6791 to (-62.38, -28.93, -199.28) mm, rotated rx 81.04 ry 30.21 rz 20.91 deg; joints [-4.035, -7.938, 68.4, 103.99, 105.779, 55.411, -153.967]
  MoveL 6792 to (-61.89, -29.05, -199.2) mm, rotated rx 81.04 ry 30.21 rz 20.91 deg; joints [-4.049, -7.959, 68.426, 103.976, 105.788, 55.407, -153.967]
  MoveL 6793 to (-61.4, -29.17, -199.11) mm, rotated rx 81.04 ry 30.21 rz 20.91 deg; joints [-4.063, -7.981, 68.454, 103.963, 105.796, 55.403, -153.967]
  MoveL 6794 to (-60.9, -29.28, -199.04) mm, rotated rx 81.04 ry 30.21 rz 20.91 deg; joints [-4.078, -8.002, 68.48, 103.949, 105.804, 55.399, -153.967]
  MoveL 6795 to (-60.38, -29.37, -199.01) mm, rotated rx 81.04 ry 30.21 rz 20.91 deg; joints [-4.094, -8.019, 68.503, 103.934, 105.813, 55.395, -153.967]
  MoveL 6796 to (-59.86, -29.44, -199) mm, rotated rx 81.04 ry 30.21 rz 20.91 deg; joints [-4.11, -8.035, 68.525, 103.919, 105.822, 55.392, -153.967]
  MoveL 6797 to (-57.33, -29.8, -198.99) mm, rotated rx 81.04 ry 30.21 rz 20.91 deg; joints [-4.188, -8.11, 68.624, 103.847, 105.866, 55.377, -153.967]
  MoveL 6798 to (-56.96, -29.91, -198.97) mm, rotated rx 81.04 ry 30.21 rz 20.91 deg; joints [-4.2, -8.123, 68.638, 103.837, 105.871, 55.377, -153.967]
  MoveL 6799 to (-56.81, -29.98, -198.85) mm, rotated rx 81.04 ry 30.21 rz 20.91 deg; joints [-4.203, -8.136, 68.655, 103.833, 105.874, 55.374, -153.967]
  MoveL 6800 to (-56.89, -29.95, -198.62) mm, rotated rx 81.04 ry 30.21 rz 20.91 deg; joints [-4.198, -8.151, 68.68, 103.835, 105.874, 55.362, -153.967]
  MoveL 6801 to (-57.22, -29.82, -198.26) mm, rotated rx 81.04 ry 30.21 rz 20.91 deg; joints [-4.183, -8.167, 68.716, 103.841, 105.872, 55.34, -153.967]
  MoveL 6802 to (-57.01, -30.56, -197.52) mm, rotated rx 81.04 ry 30.21 rz 20.91 deg; joints [-4.181, -8.235, 68.778, 103.845, 105.869, 55.346, -153.967]
  MoveL 6803 to (-55.41, -31.95, -197.5) mm, rotated rx 81.04 ry 30.21 rz 20.91 deg; joints [-4.23, -8.296, 68.783, 103.819, 105.879, 55.409, -153.967]
  MoveL 6804 to (-53.79, -33.41, -197.37) mm, rotated rx 81.04 ry 30.21 rz 20.91 deg; joints [-4.279, -8.367, 68.799, 103.793, 105.889, 55.471, -153.967]
  MoveL 6805 to (-52.11, -34.95, -197.11) mm, rotated rx 81.04 ry 30.21 rz 20.91 deg; joints [-4.328, -8.45, 68.828, 103.767, 105.9, 55.531, -153.967]
  MoveL 6806 to (-50.54, -36.37, -196.98) mm, rotated rx 81.04 ry 30.21 rz 20.91 deg; joints [-4.375, -8.519, 68.844, 103.743, 105.91, 55.591, -153.967]
  MoveL 6807 to (-49.02, -37.74, -196.72) mm, rotated rx 81.04 ry 30.21 rz 20.91 deg; joints [-4.419, -8.595, 68.874, 103.719, 105.92, 55.643, -153.967]
  MoveL 6808 to (-47.47, -39.16, -196.36) mm, rotated rx 81.04 ry 30.21 rz 20.91 deg; joints [-4.463, -8.68, 68.914, 103.694, 105.931, 55.693, -153.967]
  MoveL 6809 to (-45.86, -40.58, -196.22) mm, rotated rx 81.04 ry 30.21 rz 20.91 deg; joints [-4.511, -8.75, 68.931, 103.669, 105.942, 55.753, -153.967]
  MoveL 6810 to (-44.27, -41.97, -196.12) mm, rotated rx 81.04 ry 30.21 rz 20.91 deg; joints [-4.559, -8.816, 68.942, 103.644, 105.952, 55.814, -153.967]
  MoveL 6811 to (-42.65, -43.39, -195.98) mm, rotated rx 81.04 ry 30.21 rz 20.91 deg; joints [-4.608, -8.886, 68.959, 103.619, 105.963, 55.874, -153.967]
  MoveL 6812 to (-41.1, -44.79, -195.69) mm, rotated rx 81.04 ry 30.21 rz 20.91 deg; joints [-4.652, -8.965, 68.991, 103.595, 105.973, 55.927, -153.967]
  MoveL 6813 to (-39.42, -46.19, -195.35) mm, rotated rx 81.04 ry 30.21 rz 20.91 deg; joints [-4.7, -9.05, 69.033, 103.567, 105.987, 55.976, -153.967]
  MoveL 6814 to (-37.81, -47.57, -195.17) mm, rotated rx 81.04 ry 30.21 rz 20.91 deg; joints [-4.748, -9.122, 69.055, 103.541, 105.998, 56.033, -153.967]
  MoveL 6815 to (-36.19, -48.97, -195.06) mm, rotated rx 81.04 ry 30.21 rz 20.91 deg; joints [-4.797, -9.189, 69.066, 103.516, 106.009, 56.094, -153.967]
  MoveL 6816 to (-34.58, -50.36, -194.99) mm, rotated rx 81.04 ry 30.21 rz 20.91 deg; joints [-4.845, -9.253, 69.074, 103.491, 106.02, 56.157, -153.967]
  MoveL 6817 to (-32.94, -51.74, -194.76) mm, rotated rx 81.04 ry 30.21 rz 20.91 deg; joints [-4.893, -9.328, 69.1, 103.465, 106.032, 56.213, -153.967]
  MoveL 6818 to (-31.33, -53.12, -194.63) mm, rotated rx 81.04 ry 30.21 rz 20.91 deg; joints [-4.942, -9.396, 69.115, 103.44, 106.043, 56.272, -153.967]
  MoveL 6819 to (-29.7, -54.51, -194.55) mm, rotated rx 81.04 ry 30.21 rz 20.91 deg; joints [-4.991, -9.46, 69.122, 103.415, 106.054, 56.336, -153.967]
  MoveL 6820 to (-28.06, -55.87, -194.32) mm, rotated rx 81.04 ry 30.21 rz 20.91 deg; joints [-5.039, -9.534, 69.149, 103.389, 106.066, 56.39, -153.967]
  MoveL 6821 to (-26.4, -57.24, -194.09) mm, rotated rx 81.04 ry 30.21 rz 20.91 deg; joints [-5.087, -9.61, 69.176, 103.362, 106.079, 56.445, -153.967]
  MoveL 6822 to (-24.73, -58.64, -193.94) mm, rotated rx 81.04 ry 30.21 rz 20.91 deg; joints [-5.137, -9.68, 69.193, 103.336, 106.091, 56.505, -153.967]
  MoveL 6823 to (-23.27, -59.82, -193.81) mm, rotated rx 81.04 ry 30.21 rz 20.91 deg; joints [-5.18, -9.74, 69.208, 103.312, 106.102, 56.556, -153.967]
  MoveL 6824 to (-21.96, -60.81, -193.6) mm, rotated rx 81.04 ry 30.21 rz 20.91 deg; joints [-5.218, -9.801, 69.237, 103.29, 106.114, 56.592, -153.967]
  MoveL 6825 to (-20.77, -61.61, -193.28) mm, rotated rx 81.04 ry 30.21 rz 20.91 deg; joints [-5.251, -9.864, 69.284, 103.267, 106.126, 56.613, -153.967]
  MoveL 6826 to (-21.72, -60.48, -192.32) mm, rotated rx 81.04 ry 30.21 rz 20.91 deg; joints [-5.211, -9.897, 69.417, 103.272, 106.13, 56.506, -153.967]
  MoveL 6827 to (-21.35, -60.81, -192.32) mm, rotated rx 81.04 ry 30.21 rz 20.91 deg; joints [-5.223, -9.91, 69.416, 103.266, 106.132, 56.522, -153.967]
  MoveL 6828 to (-21, -61.16, -192.32) mm, rotated rx 81.04 ry 30.21 rz 20.91 deg; joints [-5.233, -9.924, 69.413, 103.262, 106.133, 56.54, -153.967]
  MoveL 6829 to (-20.7, -61.61, -192.29) mm, rotated rx 81.04 ry 30.21 rz 20.91 deg; joints [-5.242, -9.938, 69.405, 103.261, 106.133, 56.564, -153.967]
  MoveL 6830 to (-20.44, -62.1, -192.25) mm, rotated rx 81.04 ry 30.21 rz 20.91 deg; joints [-5.25, -9.953, 69.395, 103.262, 106.131, 56.59, -153.967]
  MoveL 6831 to (-20.21, -62.67, -192.2) mm, rotated rx 81.04 ry 30.21 rz 20.91 deg; joints [-5.256, -9.969, 69.382, 103.265, 106.127, 56.621, -153.967]
  MoveL 6832 to (-20.02, -63.22, -192.16) mm, rotated rx 81.04 ry 30.21 rz 20.91 deg; joints [-5.261, -9.982, 69.365, 103.269, 106.123, 56.652, -153.967]
  MoveL 6833 to (-19.86, -63.76, -192.14) mm, rotated rx 81.04 ry 30.21 rz 20.91 deg; joints [-5.265, -9.993, 69.345, 103.274, 106.118, 56.683, -153.967]
  MoveL 6834 to (-19.73, -64.26, -192.14) mm, rotated rx 81.04 ry 30.21 rz 20.91 deg; joints [-5.269, -10.002, 69.324, 103.279, 106.113, 56.714, -153.967]
  MoveL 6835 to (-19.58, -64.77, -192.14) mm, rotated rx 81.04 ry 30.21 rz 20.91 deg; joints [-5.274, -10.011, 69.304, 103.284, 106.108, 56.744, -153.967]
  MoveL 6836 to (-19.4, -65.33, -192.09) mm, rotated rx 81.04 ry 30.21 rz 20.91 deg; joints [-5.279, -10.024, 69.287, 103.289, 106.104, 56.776, -153.967]
  MoveL 6837 to (-19.16, -65.95, -192.01) mm, rotated rx 81.04 ry 30.21 rz 20.91 deg; joints [-5.285, -10.043, 69.275, 103.292, 106.1, 56.808, -153.967]
  MoveL 6838 to (-19, -66.44, -191.96) mm, rotated rx 81.04 ry 30.21 rz 20.91 deg; joints [-5.289, -10.056, 69.261, 103.296, 106.096, 56.835, -153.967]
  MoveL 6839 to (-18.87, -66.84, -191.93) mm, rotated rx 81.04 ry 30.21 rz 20.91 deg; joints [-5.292, -10.065, 69.248, 103.3, 106.092, 56.858, -153.967]
  MoveL 6840 to (-18.74, -67.31, -191.92) mm, rotated rx 81.04 ry 30.21 rz 20.91 deg; joints [-5.296, -10.074, 69.23, 103.304, 106.088, 56.885, -153.967]
  MoveL 6841 to (-18.6, -67.81, -191.92) mm, rotated rx 81.04 ry 30.21 rz 20.91 deg; joints [-5.3, -10.083, 69.21, 103.309, 106.083, 56.916, -153.967]
  MoveL 6842 to (-18.46, -68.29, -191.9) mm, rotated rx 81.04 ry 30.21 rz 20.91 deg; joints [-5.304, -10.092, 69.191, 103.314, 106.079, 56.944, -153.967]
  MoveL 6843 to (-18.31, -68.77, -191.88) mm, rotated rx 81.04 ry 30.21 rz 20.91 deg; joints [-5.308, -10.103, 69.176, 103.318, 106.075, 56.972, -153.967]
  MoveL 6844 to (-18.17, -69.26, -191.87) mm, rotated rx 81.04 ry 30.21 rz 20.91 deg; joints [-5.312, -10.112, 69.157, 103.322, 106.07, 57.001, -153.967]
  MoveL 6845 to (-17.47, -71.8, -191.86) mm, rotated rx 81.04 ry 30.21 rz 20.91 deg; joints [-5.332, -10.155, 69.05, 103.348, 106.046, 57.155, -153.967]
  MoveL 6846 to (-17.16, -73.22, -191.95) mm, rotated rx 81.04 ry 30.21 rz 20.91 deg; joints [-5.342, -10.171, 68.976, 103.364, 106.03, 57.246, -153.967]
  MoveL 6847 to (-17.03, -74.41, -192.2) mm, rotated rx 81.04 ry 30.21 rz 20.91 deg; joints [-5.348, -10.166, 68.887, 103.383, 106.014, 57.333, -153.967]
  MoveL 6848 to (-17.11, -75.38, -192.61) mm, rotated rx 81.04 ry 30.21 rz 20.91 deg; joints [-5.35, -10.143, 68.781, 103.405, 105.996, 57.416, -153.967]
  MoveL 6849 to (-17.38, -76.11, -193.2) mm, rotated rx 81.04 ry 30.21 rz 20.91 deg; joints [-5.348, -10.099, 68.659, 103.428, 105.976, 57.495, -153.967]
  MoveL 6850 to (-17.84, -76.63, -193.95) mm, rotated rx 81.04 ry 30.21 rz 20.91 deg; joints [-5.341, -10.036, 68.521, 103.454, 105.956, 57.571, -153.967]
  MoveL 6851 to (-18.5, -76.91, -194.86) mm, rotated rx 81.04 ry 30.21 rz 20.91 deg; joints [-5.331, -9.953, 68.366, 103.483, 105.933, 57.642, -153.967]
  MoveL 6852 to (-20.42, -76.81, -197.19) mm, rotated rx 81.04 ry 30.21 rz 20.91 deg; joints [-5.298, -9.728, 68.006, 103.547, 105.885, 57.774, -153.967]
  MoveL 6853 to (-22.52, -75.93, -199.54) mm, rotated rx 81.04 ry 30.21 rz 20.91 deg; joints [-5.259, -9.489, 67.677, 103.604, 105.844, 57.86, -153.967]
  MoveL 6854 to (-24.21, -74.42, -201.24) mm, rotated rx 81.04 ry 30.21 rz 20.91 deg; joints [-5.227, -9.303, 67.477, 103.634, 105.824, 57.87, -153.967]
  MoveL 6855 to (-24.9, -73.43, -201.86) mm, rotated rx 81.04 ry 30.21 rz 20.91 deg; joints [-5.213, -9.23, 67.426, 103.639, 105.823, 57.846, -153.967]
  MoveL 6856 to (-25.49, -72.27, -202.31) mm, rotated rx 81.04 ry 30.21 rz 20.91 deg; joints [-5.201, -9.17, 67.408, 103.638, 105.826, 57.802, -153.967]
  MoveL 6857 to (-26.36, -69.49, -202.74) mm, rotated rx 81.04 ry 30.21 rz 20.91 deg; joints [-5.18, -9.089, 67.469, 103.616, 105.849, 57.656, -153.967]
  MoveL 6858 to (-26.57, -68.5, -202.78) mm, rotated rx 81.04 ry 30.21 rz 20.91 deg; joints [-5.174, -9.072, 67.509, 103.604, 105.859, 57.598, -153.967]
  MoveL 6859 to (-26.93, -65.91, -202.78) mm, rotated rx 81.04 ry 30.21 rz 20.91 deg; joints [-5.164, -9.039, 67.635, 103.569, 105.892, 57.436, -153.967]
  MoveL 6860 to (-27.11, -64.92, -202.84) mm, rotated rx 81.04 ry 30.21 rz 20.91 deg; joints [-5.16, -9.021, 67.673, 103.556, 105.903, 57.378, -153.967]
  MoveL 6861 to (-27.26, -63.87, -202.84) mm, rotated rx 81.04 ry 30.21 rz 20.91 deg; joints [-5.156, -9.007, 67.723, 103.542, 105.916, 57.313, -153.967]
  MoveL 6862 to (-27.33, -63.4, -202.85) mm, rotated rx 81.04 ry 30.21 rz 20.91 deg; joints [-5.154, -9, 67.745, 103.536, 105.921, 57.284, -153.967]
  MoveL 6863 to (-27.41, -62.98, -202.87) mm, rotated rx 81.04 ry 30.21 rz 20.91 deg; joints [-5.152, -8.992, 67.761, 103.531, 105.926, 57.26, -153.967]
  MoveL 6864 to (-27.48, -62.52, -202.88) mm, rotated rx 81.04 ry 30.21 rz 20.91 deg; joints [-5.15, -8.985, 67.781, 103.525, 105.931, 57.232, -153.967]
  MoveL 6865 to (-27.85, -59.93, -202.89) mm, rotated rx 81.04 ry 30.21 rz 20.91 deg; joints [-5.14, -8.95, 67.903, 103.489, 105.963, 57.072, -153.967]
  MoveL 6866 to (-27.93, -59.44, -202.91) mm, rotated rx 81.04 ry 30.21 rz 20.91 deg; joints [-5.138, -8.942, 67.923, 103.483, 105.969, 57.042, -153.967]
  MoveL 6867 to (-28.04, -58.99, -202.94) mm, rotated rx 81.04 ry 30.21 rz 20.91 deg; joints [-5.135, -8.932, 67.938, 103.478, 105.973, 57.017, -153.967]
  MoveL 6868 to (-28.17, -58.57, -202.98) mm, rotated rx 81.04 ry 30.21 rz 20.91 deg; joints [-5.132, -8.921, 67.95, 103.475, 105.977, 56.994, -153.967]
  MoveL 6869 to (-28.33, -58.16, -203.02) mm, rotated rx 81.04 ry 30.21 rz 20.91 deg; joints [-5.128, -8.91, 67.96, 103.473, 105.979, 56.972, -153.967]
  MoveL 6870 to (-28.55, -57.78, -203.03) mm, rotated rx 81.04 ry 30.21 rz 20.91 deg; joints [-5.121, -8.899, 67.969, 103.472, 105.981, 56.952, -153.967]
  MoveL 6871 to (-28.81, -57.42, -203.04) mm, rotated rx 81.04 ry 30.21 rz 20.91 deg; joints [-5.113, -8.888, 67.976, 103.474, 105.981, 56.932, -153.967]
  MoveL 6872 to (-28.48, -58.11, -203.78) mm, rotated rx 81.04 ry 30.21 rz 20.91 deg; joints [-5.132, -8.849, 67.863, 103.479, 105.973, 57.009, -153.967]
  MoveL 6873 to (-29.61, -57.22, -204.33) mm, rotated rx 81.04 ry 30.21 rz 20.91 deg; joints [-5.103, -8.769, 67.793, 103.5, 105.961, 56.995, -153.967]
  MoveL 6874 to (-30.77, -56.19, -204.75) mm, rotated rx 81.04 ry 30.21 rz 20.91 deg; joints [-5.072, -8.696, 67.745, 103.518, 105.952, 56.966, -153.967]
  MoveL 6875 to (-32.03, -54.95, -205.06) mm, rotated rx 81.04 ry 30.21 rz 20.91 deg; joints [-5.037, -8.626, 67.718, 103.536, 105.944, 56.919, -153.967]
  MoveL 6876 to (-33.41, -53.47, -205.25) mm, rotated rx 81.04 ry 30.21 rz 20.91 deg; joints [-4.997, -8.56, 67.712, 103.552, 105.938, 56.853, -153.967]
  MoveL 6877 to (-34.84, -51.93, -205.44) mm, rotated rx 81.04 ry 30.21 rz 20.91 deg; joints [-4.956, -8.492, 67.706, 103.569, 105.932, 56.784, -153.967]
  MoveL 6878 to (-36.27, -50.36, -205.56) mm, rotated rx 81.04 ry 30.21 rz 20.91 deg; joints [-4.913, -8.428, 67.712, 103.585, 105.927, 56.71, -153.967]
  MoveL 6879 to (-37.72, -48.78, -205.79) mm, rotated rx 81.04 ry 30.21 rz 20.91 deg; joints [-4.872, -8.356, 67.702, 103.601, 105.921, 56.641, -153.967]
  MoveL 6880 to (-39.15, -47.2, -205.9) mm, rotated rx 81.04 ry 30.21 rz 20.91 deg; joints [-4.829, -8.292, 67.707, 103.617, 105.916, 56.566, -153.967]
  MoveL 6881 to (-40.58, -45.62, -206.02) mm, rotated rx 81.04 ry 30.21 rz 20.91 deg; joints [-4.787, -8.228, 67.711, 103.634, 105.912, 56.492, -153.967]
  MoveL 6882 to (-42, -44.03, -206.13) mm, rotated rx 81.04 ry 30.21 rz 20.91 deg; joints [-4.744, -8.163, 67.715, 103.65, 105.907, 56.417, -153.967]
  MoveL 6883 to (-43.43, -42.44, -206.37) mm, rotated rx 81.04 ry 30.21 rz 20.91 deg; joints [-4.703, -8.09, 67.704, 103.666, 105.901, 56.349, -153.967]
  MoveL 6884 to (-44.85, -40.85, -206.49) mm, rotated rx 81.04 ry 30.21 rz 20.91 deg; joints [-4.661, -8.025, 67.708, 103.683, 105.897, 56.274, -153.967]
  MoveL 6885 to (-46.27, -39.37, -206.59) mm, rotated rx 81.04 ry 30.21 rz 20.91 deg; joints [-4.619, -7.963, 67.708, 103.7, 105.891, 56.206, -153.967]
  MoveL 6886 to (-47.73, -37.98, -206.8) mm, rotated rx 81.04 ry 30.21 rz 20.91 deg; joints [-4.576, -7.892, 67.688, 103.722, 105.882, 56.15, -153.967]
  MoveL 6887 to (-49.38, -36.1, -206.94) mm, rotated rx 81.04 ry 30.21 rz 20.91 deg; joints [-4.527, -7.816, 67.693, 103.74, 105.877, 56.062, -153.967]
  MoveL 6888 to (-50.9, -34.18, -207.02) mm, rotated rx 81.04 ry 30.21 rz 20.91 deg; joints [-4.481, -7.747, 67.712, 103.754, 105.876, 55.967, -153.967]
  MoveL 6889 to (-52.36, -32.42, -207.05) mm, rotated rx 81.04 ry 30.21 rz 20.91 deg; joints [-4.437, -7.684, 67.73, 103.769, 105.873, 55.88, -153.967]
  MoveL 6890 to (-53.72, -30.88, -207.1) mm, rotated rx 81.04 ry 30.21 rz 20.91 deg; joints [-4.395, -7.626, 67.741, 103.784, 105.87, 55.805, -153.967]
  MoveL 6891 to (-55.02, -29.41, -207.22) mm, rotated rx 81.04 ry 30.21 rz 20.91 deg; joints [-4.356, -7.565, 67.741, 103.799, 105.866, 55.738, -153.967]
  MoveL 6892 to (-56.36, -27.89, -207.28) mm, rotated rx 81.04 ry 30.21 rz 20.91 deg; joints [-4.316, -7.506, 67.748, 103.815, 105.862, 55.667, -153.967]
  MoveL 6893 to (-57.77, -26.3, -207.35) mm, rotated rx 81.04 ry 30.21 rz 20.91 deg; joints [-4.273, -7.443, 67.755, 103.832, 105.858, 55.591, -153.967]
  MoveL 6894 to (-59.07, -24.79, -207.53) mm, rotated rx 81.04 ry 30.21 rz 20.91 deg; joints [-4.235, -7.376, 67.748, 103.847, 105.854, 55.526, -153.967]
  MoveL 6895 to (-60.3, -23.34, -207.85) mm, rotated rx 81.04 ry 30.21 rz 20.91 deg; joints [-4.201, -7.302, 67.725, 103.861, 105.85, 55.47, -153.967]
  MoveL 6896 to (-60.45, -22.48, -208.89) mm, rotated rx 81.04 ry 30.21 rz 20.91 deg; joints [-4.208, -7.211, 67.632, 103.856, 105.853, 55.473, -153.967]
  MoveL 6897 to (-60.24, -22.63, -209.41) mm, rotated rx 81.04 ry 30.21 rz 20.91 deg; joints [-4.221, -7.18, 67.57, 103.854, 105.852, 55.506, -153.967]
  MoveL 6898 to (-60.22, -22.63, -209.73) mm, rotated rx 81.04 ry 30.21 rz 20.91 deg; joints [-4.225, -7.157, 67.531, 103.854, 105.85, 55.522, -153.967]
  MoveL 6899 to (-60.37, -22.48, -209.89) mm, rotated rx 81.04 ry 30.21 rz 20.91 deg; joints [-4.222, -7.139, 67.512, 103.857, 105.848, 55.523, -153.967]
  MoveL 6900 to (-60.72, -22.24, -209.93) mm, rotated rx 81.04 ry 30.21 rz 20.91 deg; joints [-4.212, -7.123, 67.503, 103.864, 105.845, 55.516, -153.967]
  MoveL 6901 to (-61.18, -21.99, -209.95) mm, rotated rx 81.04 ry 30.21 rz 20.91 deg; joints [-4.198, -7.106, 67.492, 103.874, 105.839, 55.508, -153.967]
  MoveL 6902 to (-61.74, -21.78, -209.96) mm, rotated rx 81.04 ry 30.21 rz 20.91 deg; joints [-4.181, -7.087, 67.475, 103.888, 105.832, 55.504, -153.967]
  MoveL 6903 to (-62.34, -21.59, -209.97) mm, rotated rx 81.04 ry 30.21 rz 20.91 deg; joints [-4.162, -7.068, 67.455, 103.903, 105.823, 55.502, -153.967]
  MoveL 6904 to (-65.89, -20.68, -209.97) mm, rotated rx 81.04 ry 30.21 rz 20.91 deg; joints [-4.052, -6.957, 67.334, 103.998, 105.767, 55.499, -153.967]
  MoveL 6905 to (-66.31, -20.56, -210) mm, rotated rx 81.04 ry 30.21 rz 20.91 deg; joints [-4.039, -6.942, 67.317, 104.01, 105.761, 55.499, -153.967]
  MoveL 6906 to (-66.78, -20.43, -210.01) mm, rotated rx 81.04 ry 30.21 rz 20.91 deg; joints [-4.025, -6.927, 67.3, 104.022, 105.753, 55.499, -153.967]
  MoveL 6907 to (-67.28, -20.3, -210.01) mm, rotated rx 81.04 ry 30.21 rz 20.91 deg; joints [-4.009, -6.91, 67.282, 104.036, 105.746, 55.498, -153.967]
  MoveL 6908 to (-67.76, -20.16, -210.03) mm, rotated rx 81.04 ry 30.21 rz 20.91 deg; joints [-3.995, -6.894, 67.264, 104.048, 105.738, 55.498, -153.967]
  MoveL 6909 to (-68.2, -20.02, -210.07) mm, rotated rx 81.04 ry 30.21 rz 20.91 deg; joints [-3.981, -6.877, 67.246, 104.06, 105.731, 55.498, -153.967]
  MoveL 6910 to (-68.6, -19.88, -210.13) mm, rotated rx 81.04 ry 30.21 rz 20.91 deg; joints [-3.97, -6.86, 67.227, 104.07, 105.725, 55.498, -153.967]
  MoveL 6911 to (-69.05, -19.73, -210.16) mm, rotated rx 81.04 ry 30.21 rz 20.91 deg; joints [-3.956, -6.843, 67.208, 104.082, 105.719, 55.498, -153.967]
  MoveL 6912 to (-69.52, -19.6, -210.18) mm, rotated rx 81.04 ry 30.21 rz 20.91 deg; joints [-3.942, -6.827, 67.19, 104.094, 105.711, 55.498, -153.967]
  MoveL 6913 to (-70.01, -19.47, -210.19) mm, rotated rx 81.04 ry 30.21 rz 20.91 deg; joints [-3.927, -6.811, 67.173, 104.107, 105.704, 55.498, -153.967]
  MoveL 6914 to (-70.52, -19.34, -210.19) mm, rotated rx 81.04 ry 30.21 rz 20.91 deg; joints [-3.911, -6.795, 67.155, 104.121, 105.696, 55.498, -153.967]
  MoveL 6915 to (-73.26, -18.34, -210.53) mm, rotated rx 81.04 ry 30.21 rz 20.91 deg; joints [-3.83, -6.68, 67.032, 104.191, 105.655, 55.496, -153.967]
  MoveL 6916 to (-74.38, -17.68, -210.96) mm, rotated rx 81.04 ry 30.21 rz 20.91 deg; joints [-3.8, -6.609, 66.957, 104.216, 105.64, 55.495, -153.967]
  MoveL 6917 to (-75.33, -16.91, -211.57) mm, rotated rx 81.04 ry 30.21 rz 20.91 deg; joints [-3.778, -6.527, 66.874, 104.235, 105.629, 55.495, -153.967]
  MoveL 6918 to (-76.74, -15.05, -213.3) mm, rotated rx 81.04 ry 30.21 rz 20.91 deg; joints [-3.755, -6.337, 66.682, 104.255, 105.617, 55.493, -153.967]
  MoveL 6919 to (-77.47, -12.77, -215.72) mm, rotated rx 81.04 ry 30.21 rz 20.91 deg; joints [-3.761, -6.108, 66.455, 104.25, 105.62, 55.492, -153.967]
  MoveL 6920 to (-77.46, -10.73, -218.15) mm, rotated rx 81.04 ry 30.21 rz 20.91 deg; joints [-3.79, -5.903, 66.25, 104.225, 105.634, 55.496, -153.967]
  MoveL 6921 to (-77.14, -10.06, -219.1) mm, rotated rx 81.04 ry 30.21 rz 20.91 deg; joints [-3.811, -5.833, 66.179, 104.208, 105.644, 55.5, -153.967]
  MoveL 6922 to (-76.61, -9.61, -219.88) mm, rotated rx 81.04 ry 30.21 rz 20.91 deg; joints [-3.837, -5.785, 66.128, 104.187, 105.656, 55.506, -153.967]
  MoveL 6923 to (-76.26, -9.48, -220.2) mm, rotated rx 81.04 ry 30.21 rz 20.91 deg; joints [-3.851, -5.769, 66.11, 104.176, 105.662, 55.509, -153.967]
  MoveL 6924 to (-75.86, -9.4, -220.48) mm, rotated rx 81.04 ry 30.21 rz 20.91 deg; joints [-3.867, -5.758, 66.097, 104.163, 105.669, 55.513, -153.967]
  MoveL 6925 to (-74.91, -9.41, -220.92) mm, rotated rx 81.04 ry 30.21 rz 20.91 deg; joints [-3.902, -5.753, 66.088, 104.135, 105.685, 55.522, -153.967]
  MoveL 6926 to (-73.75, -9.65, -221.17) mm, rotated rx 81.04 ry 30.21 rz 20.91 deg; joints [-3.941, -5.77, 66.099, 104.104, 105.702, 55.532, -153.967]
  MoveL 6927 to (-72.38, -10.12, -221.26) mm, rotated rx 81.04 ry 30.21 rz 20.91 deg; joints [-3.984, -5.808, 66.131, 104.07, 105.722, 55.544, -153.967]
  MoveL 6928 to (-71.89, -10.31, -221.26) mm, rotated rx 81.04 ry 30.21 rz 20.91 deg; joints [-3.999, -5.824, 66.145, 104.058, 105.729, 55.548, -153.967]
  MoveL 6929 to (-71.48, -10.5, -221.23) mm, rotated rx 81.04 ry 30.21 rz 20.91 deg; joints [-4.012, -5.84, 66.159, 104.048, 105.734, 55.551, -153.967]
  MoveL 6930 to (-71.09, -10.69, -221.19) mm, rotated rx 81.04 ry 30.21 rz 20.91 deg; joints [-4.023, -5.857, 66.174, 104.039, 105.739, 55.554, -153.967]
  MoveL 6931 to (-70.72, -10.89, -221.13) mm, rotated rx 81.04 ry 30.21 rz 20.91 deg; joints [-4.034, -5.874, 66.19, 104.03, 105.744, 55.557, -153.967]
  MoveL 6932 to (-70.31, -11.08, -221.09) mm, rotated rx 81.04 ry 30.21 rz 20.91 deg; joints [-4.046, -5.891, 66.205, 104.02, 105.749, 55.561, -153.967]
  MoveL 6933 to (-69.84, -11.28, -221.07) mm, rotated rx 81.04 ry 30.21 rz 20.91 deg; joints [-4.061, -5.908, 66.22, 104.009, 105.756, 55.565, -153.967]
  MoveL 6934 to (-69.35, -11.47, -221.07) mm, rotated rx 81.04 ry 30.21 rz 20.91 deg; joints [-4.076, -5.924, 66.234, 103.997, 105.762, 55.569, -153.967]
  MoveL 6935 to (-68.89, -11.66, -221.07) mm, rotated rx 81.04 ry 30.21 rz 20.91 deg; joints [-4.09, -5.94, 66.247, 103.986, 105.769, 55.573, -153.967]
  MoveL 6936 to (-68.46, -11.84, -221.04) mm, rotated rx 81.04 ry 30.21 rz 20.91 deg; joints [-4.103, -5.956, 66.262, 103.975, 105.775, 55.576, -153.967]
  MoveL 6937 to (-68.07, -12.03, -220.99) mm, rotated rx 81.04 ry 30.21 rz 20.91 deg; joints [-4.114, -5.973, 66.278, 103.966, 105.78, 55.579, -153.967]
  MoveL 6938 to (-67.69, -12.21, -220.93) mm, rotated rx 81.04 ry 30.21 rz 20.91 deg; joints [-4.125, -5.99, 66.294, 103.957, 105.785, 55.581, -153.967]
  MoveL 6939 to (-67.27, -12.42, -220.87) mm, rotated rx 81.04 ry 30.21 rz 20.91 deg; joints [-4.138, -6.009, 66.311, 103.947, 105.791, 55.584, -153.967]
  MoveL 6940 to (-66.71, -12.67, -220.84) mm, rotated rx 81.04 ry 30.21 rz 20.91 deg; joints [-4.155, -6.03, 66.33, 103.934, 105.798, 55.589, -153.967]
  MoveL 6941 to (-65.99, -12.98, -220.82) mm, rotated rx 81.04 ry 30.21 rz 20.91 deg; joints [-4.177, -6.056, 66.352, 103.916, 105.808, 55.596, -153.967]
  MoveL 6942 to (-64.53, -13.56, -220.82) mm, rotated rx 81.04 ry 30.21 rz 20.91 deg; joints [-4.222, -6.104, 66.392, 103.881, 105.828, 55.609, -153.967]
  MoveL 6943 to (-63.76, -13.88, -220.79) mm, rotated rx 81.04 ry 30.21 rz 20.91 deg; joints [-4.246, -6.132, 66.417, 103.862, 105.838, 55.615, -153.967]
  MoveL 6944 to (-63.18, -14.13, -220.77) mm, rotated rx 81.04 ry 30.21 rz 20.91 deg; joints [-4.263, -6.152, 66.433, 103.848, 105.846, 55.621, -153.967]
  MoveL 6945 to (-62.75, -14.35, -220.77) mm, rotated rx 81.04 ry 30.21 rz 20.91 deg; joints [-4.277, -6.168, 66.444, 103.838, 105.851, 55.628, -153.967]
  MoveL 6946 to (-62.39, -14.58, -220.74) mm, rotated rx 81.04 ry 30.21 rz 20.91 deg; joints [-4.287, -6.182, 66.452, 103.831, 105.855, 55.635, -153.967]
  MoveL 6947 to (-62.25, -14.72, -220.64) mm, rotated rx 81.04 ry 30.21 rz 20.91 deg; joints [-4.291, -6.196, 66.465, 103.829, 105.856, 55.636, -153.967]
  MoveL 6948 to (-62.32, -14.73, -220.42) mm, rotated rx 81.04 ry 30.21 rz 20.91 deg; joints [-4.286, -6.21, 66.489, 103.83, 105.856, 55.626, -153.967]
  MoveL 6949 to (-62.62, -14.57, -220.07) mm, rotated rx 81.04 ry 30.21 rz 20.91 deg; joints [-4.273, -6.226, 66.527, 103.835, 105.855, 55.602, -153.967]
  MoveL 6950 to (-62.67, -15.35, -219.37) mm, rotated rx 81.04 ry 30.21 rz 20.91 deg; joints [-4.263, -6.286, 66.575, 103.847, 105.847, 55.614, -153.967]
  MoveL 6951 to (-61.57, -17.03, -219.22) mm, rotated rx 81.04 ry 30.21 rz 20.91 deg; joints [-4.295, -6.348, 66.562, 103.84, 105.845, 55.693, -153.967]
  MoveL 6952 to (-60.54, -18.65, -218.93) mm, rotated rx 81.04 ry 30.21 rz 20.91 deg; joints [-4.323, -6.417, 66.564, 103.835, 105.843, 55.763, -153.967]
  MoveL 6953 to (-59.48, -20.27, -218.66) mm, rotated rx 81.04 ry 30.21 rz 20.91 deg; joints [-4.352, -6.486, 66.567, 103.829, 105.841, 55.834, -153.967]
  MoveL 6954 to (-58.43, -21.89, -218.39) mm, rotated rx 81.04 ry 30.21 rz 20.91 deg; joints [-4.382, -6.554, 66.569, 103.823, 105.84, 55.904, -153.967]
  MoveL 6955 to (-57.31, -23.58, -218.17) mm, rotated rx 81.04 ry 30.21 rz 20.91 deg; joints [-4.414, -6.62, 66.563, 103.816, 105.838, 55.981, -153.967]
  MoveL 6956 to (-56.19, -25.38, -218.03) mm, rotated rx 81.04 ry 30.21 rz 20.91 deg; joints [-4.446, -6.682, 66.542, 103.812, 105.834, 56.069, -153.967]
  MoveL 6957 to (-54.95, -27.6, -217.92) mm, rotated rx 81.04 ry 30.21 rz 20.91 deg; joints [-4.483, -6.749, 66.5, 103.812, 105.826, 56.184, -153.967]
  MoveL 6958 to (-53.44, -29.57, -217.85) mm, rotated rx 81.04 ry 30.21 rz 20.91 deg; joints [-4.528, -6.819, 66.479, 103.799, 105.826, 56.281, -153.967]
  MoveL 6959 to (-52.15, -31.25, -217.73) mm, rotated rx 81.04 ry 30.21 rz 20.91 deg; joints [-4.567, -6.881, 66.467, 103.788, 105.827, 56.361, -153.967]
  MoveL 6960 to (-51.04, -32.78, -217.56) mm, rotated rx 81.04 ry 30.21 rz 20.91 deg; joints [-4.599, -6.942, 66.462, 103.779, 105.827, 56.432, -153.967]
  MoveL 6961 to (-49.88, -34.46, -217.43) mm, rotated rx 81.04 ry 30.21 rz 20.91 deg; joints [-4.633, -7.002, 66.445, 103.772, 105.826, 56.513, -153.967]
  MoveL 6962 to (-48.69, -36.17, -217.3) mm, rotated rx 81.04 ry 30.21 rz 20.91 deg; joints [-4.667, -7.063, 66.427, 103.765, 105.824, 56.597, -153.967]
  MoveL 6963 to (-47.46, -37.96, -217.23) mm, rotated rx 81.04 ry 30.21 rz 20.91 deg; joints [-4.704, -7.12, 66.399, 103.758, 105.822, 56.688, -153.967]
  MoveL 6964 to (-46.24, -39.71, -217) mm, rotated rx 81.04 ry 30.21 rz 20.91 deg; joints [-4.739, -7.189, 66.392, 103.751, 105.821, 56.769, -153.967]
  MoveL 6965 to (-45.02, -41.46, -216.89) mm, rotated rx 81.04 ry 30.21 rz 20.91 deg; joints [-4.775, -7.25, 66.371, 103.744, 105.82, 56.856, -153.967]
  MoveL 6966 to (-43.79, -43.21, -216.67) mm, rotated rx 81.04 ry 30.21 rz 20.91 deg; joints [-4.809, -7.318, 66.364, 103.736, 105.819, 56.937, -153.967]
  MoveL 6967 to (-42.57, -44.96, -216.56) mm, rotated rx 81.04 ry 30.21 rz 20.91 deg; joints [-4.845, -7.378, 66.341, 103.729, 105.818, 57.024, -153.967]
  MoveL 6968 to (-41.33, -46.7, -216.34) mm, rotated rx 81.04 ry 30.21 rz 20.91 deg; joints [-4.881, -7.446, 66.333, 103.721, 105.817, 57.106, -153.967]
  MoveL 6969 to (-40.1, -48.44, -216.23) mm, rotated rx 81.04 ry 30.21 rz 20.91 deg; joints [-4.917, -7.505, 66.31, 103.714, 105.816, 57.193, -153.967]
  MoveL 6970 to (-38.87, -50.19, -216.12) mm, rotated rx 81.04 ry 30.21 rz 20.91 deg; joints [-4.953, -7.564, 66.286, 103.707, 105.814, 57.281, -153.967]
  MoveL 6971 to (-37.72, -51.72, -215.89) mm, rotated rx 81.04 ry 30.21 rz 20.91 deg; joints [-4.985, -7.628, 66.286, 103.698, 105.816, 57.35, -153.967]
  MoveL 6972 to (-36.59, -53.16, -215.59) mm, rotated rx 81.04 ry 30.21 rz 20.91 deg; joints [-5.016, -7.695, 66.297, 103.688, 105.818, 57.41, -153.967]
  MoveL 6973 to (-35.43, -54.54, -215.2) mm, rotated rx 81.04 ry 30.21 rz 20.91 deg; joints [-5.046, -7.769, 66.324, 103.676, 105.822, 57.462, -153.967]
  MoveL 6974 to (-36, -53.24, -214.28) mm, rotated rx 81.04 ry 30.21 rz 20.91 deg; joints [-5.019, -7.811, 66.485, 103.666, 105.837, 57.339, -153.967]
  MoveL 6975 to (-35.8, -53.54, -214.22) mm, rotated rx 81.04 ry 30.21 rz 20.91 deg; joints [-5.025, -7.824, 66.485, 103.665, 105.836, 57.352, -153.967]
  MoveL 6976 to (-35.62, -53.87, -214.16) mm, rotated rx 81.04 ry 30.21 rz 20.91 deg; joints [-5.029, -7.836, 66.482, 103.665, 105.835, 57.368, -153.967]
  MoveL 6977 to (-35.5, -54.26, -214.13) mm, rotated rx 81.04 ry 30.21 rz 20.91 deg; joints [-5.033, -7.846, 66.471, 103.668, 105.832, 57.389, -153.967]
  MoveL 6978 to (-35.41, -54.71, -214.1) mm, rotated rx 81.04 ry 30.21 rz 20.91 deg; joints [-5.035, -7.854, 66.454, 103.673, 105.827, 57.415, -153.967]
  MoveL 6979 to (-35.37, -55.21, -214.1) mm, rotated rx 81.04 ry 30.21 rz 20.91 deg; joints [-5.036, -7.861, 66.43, 103.681, 105.82, 57.446, -153.967]
  MoveL 6980 to (-35.36, -55.72, -214.09) mm, rotated rx 81.04 ry 30.21 rz 20.91 deg; joints [-5.036, -7.866, 66.403, 103.69, 105.813, 57.479, -153.967]
  MoveL 6981 to (-35.34, -56.78, -214.09) mm, rotated rx 81.04 ry 30.21 rz 20.91 deg; joints [-5.036, -7.876, 66.347, 103.708, 105.797, 57.546, -153.967]
  MoveL 6982 to (-35.32, -57.27, -214.07) mm, rotated rx 81.04 ry 30.21 rz 20.91 deg; joints [-5.036, -7.882, 66.324, 103.716, 105.79, 57.575, -153.967]
  MoveL 6983 to (-35.28, -57.73, -214.02) mm, rotated rx 81.04 ry 30.21 rz 20.91 deg; joints [-5.037, -7.891, 66.307, 103.723, 105.784, 57.602, -153.967]
  MoveL 6984 to (-35.22, -58.25, -213.95) mm, rotated rx 81.04 ry 30.21 rz 20.91 deg; joints [-5.037, -7.904, 66.291, 103.73, 105.778, 57.63, -153.967]
  MoveL 6985 to (-35.18, -58.83, -213.88) mm, rotated rx 81.04 ry 30.21 rz 20.91 deg; joints [-5.038, -7.915, 66.27, 103.738, 105.77, 57.663, -153.967]
  MoveL 6986 to (-35.15, -59.4, -213.85) mm, rotated rx 81.04 ry 30.21 rz 20.91 deg; joints [-5.038, -7.923, 66.244, 103.748, 105.762, 57.698, -153.967]
  MoveL 6987 to (-35.13, -59.94, -213.84) mm, rotated rx 81.04 ry 30.21 rz 20.91 deg; joints [-5.038, -7.93, 66.217, 103.757, 105.754, 57.731, -153.967]
  MoveL 6988 to (-35.13, -60.48, -213.83) mm, rotated rx 81.04 ry 30.21 rz 20.91 deg; joints [-5.038, -7.935, 66.188, 103.766, 105.746, 57.766, -153.967]
  MoveL 6989 to (-35.11, -61.53, -213.83) mm, rotated rx 81.04 ry 30.21 rz 20.91 deg; joints [-5.038, -7.944, 66.132, 103.784, 105.731, 57.832, -153.967]
  MoveL 6990 to (-35.07, -62.56, -213.81) mm, rotated rx 81.04 ry 30.21 rz 20.91 deg; joints [-5.039, -7.956, 66.081, 103.801, 105.716, 57.896, -153.967]
  MoveL 6991 to (-35.03, -65.17, -213.81) mm, rotated rx 81.04 ry 30.21 rz 20.91 deg; joints [-5.038, -7.98, 65.938, 103.846, 105.676, 58.063, -153.967]
  MoveL 6992 to (-35.08, -66.62, -213.9) mm, rotated rx 81.04 ry 30.21 rz 20.91 deg; joints [-5.037, -7.984, 65.845, 103.874, 105.652, 58.161, -153.967]
  MoveL 6993 to (-35.27, -67.78, -214.16) mm, rotated rx 81.04 ry 30.21 rz 20.91 deg; joints [-5.034, -7.968, 65.738, 103.901, 105.629, 58.252, -153.967]
  MoveL 6994 to (-35.6, -68.67, -214.6) mm, rotated rx 81.04 ry 30.21 rz 20.91 deg; joints [-5.028, -7.933, 65.619, 103.928, 105.606, 58.337, -153.967]
  MoveL 6995 to (-35.81, -69, -214.88) mm, rotated rx 81.04 ry 30.21 rz 20.91 deg; joints [-5.025, -7.908, 65.554, 103.942, 105.594, 58.376, -153.967]
  MoveL 6996 to (-36.06, -69.27, -215.21) mm, rotated rx 81.04 ry 30.21 rz 20.91 deg; joints [-5.021, -7.878, 65.486, 103.956, 105.583, 58.414, -153.967]
  MoveL 6997 to (-36.66, -69.59, -216) mm, rotated rx 81.04 ry 30.21 rz 20.91 deg; joints [-5.011, -7.803, 65.34, 103.983, 105.561, 58.484, -153.967]
  MoveL 6998 to (-37.4, -69.62, -216.97) mm, rotated rx 81.04 ry 30.21 rz 20.91 deg; joints [-4.999, -7.708, 65.181, 104.01, 105.539, 58.548, -153.967]
  MoveL 6999 to (-39.3, -68.85, -219.42) mm, rotated rx 81.04 ry 30.21 rz 20.91 deg; joints [-4.969, -7.46, 64.821, 104.064, 105.496, 58.656, -153.967]
  MoveL 7000 to (-41.16, -67.29, -221.88) mm, rotated rx 81.04 ry 30.21 rz 20.91 deg; joints [-4.94, -7.206, 64.506, 104.104, 105.466, 58.713, -153.967]
  MoveL 7001 to (-42.38, -65.27, -223.63) mm, rotated rx 81.04 ry 30.21 rz 20.91 deg; joints [-4.923, -7.019, 64.334, 104.113, 105.461, 58.696, -153.967]
  MoveL 7002 to (-42.76, -64.09, -224.25) mm, rotated rx 81.04 ry 30.21 rz 20.91 deg; joints [-4.919, -6.952, 64.303, 104.107, 105.468, 58.659, -153.967]
  MoveL 7003 to (-42.97, -62.8, -224.68) mm, rotated rx 81.04 ry 30.21 rz 20.91 deg; joints [-4.918, -6.902, 64.308, 104.093, 105.48, 58.603, -153.967]
  MoveL 7004 to (-42.94, -59.87, -225.04) mm, rotated rx 81.04 ry 30.21 rz 20.91 deg; joints [-4.924, -6.852, 64.428, 104.043, 105.525, 58.434, -153.967]
  MoveL 7005 to (-42.64, -57.26, -225.03) mm, rotated rx 81.04 ry 30.21 rz 20.91 deg; joints [-4.934, -6.839, 64.587, 103.988, 105.572, 58.262, -153.967]
  MoveL 7006 to (-42.58, -56.73, -225.02) mm, rotated rx 81.04 ry 30.21 rz 20.91 deg; joints [-4.936, -6.838, 64.62, 103.977, 105.581, 58.227, -153.967]
  MoveL 7007 to (-42.5, -56.2, -224.99) mm, rotated rx 81.04 ry 30.21 rz 20.91 deg; joints [-4.938, -6.838, 64.658, 103.965, 105.591, 58.19, -153.967]
  MoveL 7008 to (-42.44, -55.7, -224.98) mm, rotated rx 81.04 ry 30.21 rz 20.91 deg; joints [-4.94, -6.836, 64.689, 103.955, 105.6, 58.157, -153.967]
  MoveL 7009 to (-42.4, -55.26, -225) mm, rotated rx 81.04 ry 30.21 rz 20.91 deg; joints [-4.942, -6.832, 64.713, 103.946, 105.608, 58.129, -153.967]
  MoveL 7010 to (-42.36, -54.77, -225.03) mm, rotated rx 81.04 ry 30.21 rz 20.91 deg; joints [-4.944, -6.827, 64.738, 103.936, 105.616, 58.099, -153.967]
  MoveL 7011 to (-42.34, -54.2, -225.1) mm, rotated rx 81.04 ry 30.21 rz 20.91 deg; joints [-4.945, -6.818, 64.762, 103.926, 105.625, 58.065, -153.967]
  MoveL 7012 to (-42.32, -53.62, -225.17) mm, rotated rx 81.04 ry 30.21 rz 20.91 deg; joints [-4.947, -6.807, 64.784, 103.916, 105.633, 58.033, -153.967]
  MoveL 7013 to (-42.29, -53.05, -225.22) mm, rotated rx 81.04 ry 30.21 rz 20.91 deg; joints [-4.949, -6.799, 64.81, 103.905, 105.643, 57.999, -153.967]
  MoveL 7014 to (-42.25, -52.52, -225.25) mm, rotated rx 81.04 ry 30.21 rz 20.91 deg; joints [-4.95, -6.794, 64.838, 103.895, 105.651, 57.966, -153.967]
  MoveL 7015 to (-42.2, -52.01, -225.26) mm, rotated rx 81.04 ry 30.21 rz 20.91 deg; joints [-4.952, -6.79, 64.868, 103.884, 105.66, 57.932, -153.967]
  MoveL 7016 to (-42.14, -51.49, -225.26) mm, rotated rx 81.04 ry 30.21 rz 20.91 deg; joints [-4.954, -6.788, 64.899, 103.873, 105.67, 57.898, -153.967]
  MoveL 7017 to (-42.1, -50.92, -225.29) mm, rotated rx 81.04 ry 30.21 rz 20.91 deg; joints [-4.956, -6.781, 64.927, 103.862, 105.679, 57.863, -153.967]
  MoveL 7018 to (-42.08, -50.37, -225.34) mm, rotated rx 81.04 ry 30.21 rz 20.91 deg; joints [-4.957, -6.773, 64.951, 103.852, 105.687, 57.831, -153.967]
  MoveL 7019 to (-42.09, -49.81, -225.41) mm, rotated rx 81.04 ry 30.21 rz 20.91 deg; joints [-4.958, -6.762, 64.972, 103.843, 105.695, 57.799, -153.967]
  MoveL 7020 to (-42.14, -49.31, -225.47) mm, rotated rx 81.04 ry 30.21 rz 20.91 deg; joints [-4.958, -6.752, 64.99, 103.836, 105.702, 57.771, -153.967]
  MoveL 7021 to (-42.23, -48.86, -225.5) mm, rotated rx 81.04 ry 30.21 rz 20.91 deg; joints [-4.955, -6.743, 65.006, 103.831, 105.706, 57.745, -153.967]
  MoveL 7022 to (-42.37, -48.48, -225.51) mm, rotated rx 81.04 ry 30.21 rz 20.91 deg; joints [-4.951, -6.735, 65.018, 103.829, 105.709, 57.724, -153.967]
  MoveL 7023 to (-42.54, -48.13, -225.51) mm, rotated rx 81.04 ry 30.21 rz 20.91 deg; joints [-4.946, -6.727, 65.03, 103.827, 105.711, 57.704, -153.967]
  MoveL 7024 to (-42.15, -49.35, -226.39) mm, rotated rx 81.04 ry 30.21 rz 20.91 deg; joints [-4.968, -6.682, 64.868, 103.842, 105.694, 57.824, -153.967]
  MoveL 7025 to (-42.98, -47.99, -226.67) mm, rotated rx 81.04 ry 30.21 rz 20.91 deg; joints [-4.946, -6.624, 64.867, 103.844, 105.697, 57.765, -153.967]
  MoveL 7026 to (-43.88, -46.42, -226.86) mm, rotated rx 81.04 ry 30.21 rz 20.91 deg; joints [-4.921, -6.57, 64.884, 103.845, 105.701, 57.689, -153.967]
  MoveL 7027 to (-44.87, -44.62, -226.99) mm, rotated rx 81.04 ry 30.21 rz 20.91 deg; joints [-4.893, -6.515, 64.918, 103.844, 105.708, 57.596, -153.967]
  MoveL 7028 to (-45.92, -42.64, -227.08) mm, rotated rx 81.04 ry 30.21 rz 20.91 deg; joints [-4.862, -6.46, 64.964, 103.841, 105.717, 57.49, -153.967]
  MoveL 7029 to (-46.93, -40.76, -227.23) mm, rotated rx 81.04 ry 30.21 rz 20.91 deg; joints [-4.833, -6.403, 64.998, 103.84, 105.724, 57.394, -153.967]
  MoveL 7030 to (-47.95, -38.88, -227.44) mm, rotated rx 81.04 ry 30.21 rz 20.91 deg; joints [-4.805, -6.34, 65.023, 103.839, 105.731, 57.302, -153.967]
  MoveL 7031 to (-48.91, -37.09, -227.57) mm, rotated rx 81.04 ry 30.21 rz 20.91 deg; joints [-4.777, -6.286, 65.057, 103.837, 105.738, 57.21, -153.967]
  MoveL 7032 to (-49.8, -35.47, -227.83) mm, rotated rx 81.04 ry 30.21 rz 20.91 deg; joints [-4.753, -6.225, 65.067, 103.838, 105.743, 57.135, -153.967]
  MoveL 7033 to (-50.78, -33.65, -228.05) mm, rotated rx 81.04 ry 30.21 rz 20.91 deg; joints [-4.726, -6.163, 65.088, 103.837, 105.749, 57.047, -153.967]
  MoveL 7034 to (-51.75, -31.81, -228.19) mm, rotated rx 81.04 ry 30.21 rz 20.91 deg; joints [-4.699, -6.106, 65.121, 103.835, 105.757, 56.953, -153.967]
  MoveL 7035 to (-52.74, -29.91, -228.29) mm, rotated rx 81.04 ry 30.21 rz 20.91 deg; joints [-4.67, -6.051, 65.16, 103.833, 105.765, 56.855, -153.967]
  MoveL 7036 to (-53.73, -28.04, -228.52) mm, rotated rx 81.04 ry 30.21 rz 20.91 deg; joints [-4.642, -5.986, 65.182, 103.832, 105.772, 56.764, -153.967]
  MoveL 7037 to (-54.71, -26.13, -228.78) mm, rotated rx 81.04 ry 30.21 rz 20.91 deg; joints [-4.616, -5.919, 65.201, 103.83, 105.779, 56.674, -153.967]
  MoveL 7038 to (-55.68, -24.24, -228.87) mm, rotated rx 81.04 ry 30.21 rz 20.91 deg; joints [-4.587, -5.865, 65.241, 103.828, 105.787, 56.575, -153.967]
  MoveL 7039 to (-56.68, -22.31, -228.91) mm, rotated rx 81.04 ry 30.21 rz 20.91 deg; joints [-4.557, -5.812, 65.287, 103.826, 105.796, 56.472, -153.967]
  MoveL 7040 to (-57.65, -20.43, -229.02) mm, rotated rx 81.04 ry 30.21 rz 20.91 deg; joints [-4.529, -5.757, 65.324, 103.824, 105.804, 56.375, -153.967]
  MoveL 7041 to (-58.61, -18.54, -229.22) mm, rotated rx 81.04 ry 30.21 rz 20.91 deg; joints [-4.502, -5.694, 65.349, 103.822, 105.812, 56.283, -153.967]
  MoveL 7042 to (-59.54, -16.68, -229.55) mm, rotated rx 81.04 ry 30.21 rz 20.91 deg; joints [-4.478, -5.621, 65.356, 103.82, 105.819, 56.2, -153.967]
  MoveL 7043 to (-60.48, -14.75, -229.81) mm, rotated rx 81.04 ry 30.21 rz 20.91 deg; joints [-4.452, -5.554, 65.375, 103.818, 105.827, 56.108, -153.967]
  MoveL 7044 to (-61.42, -12.83, -230.01) mm, rotated rx 81.04 ry 30.21 rz 20.91 deg; joints [-4.425, -5.49, 65.401, 103.815, 105.836, 56.015, -153.967]
  MoveL 7045 to (-62.37, -10.87, -230.25) mm, rotated rx 81.04 ry 30.21 rz 20.91 deg; joints [-4.399, -5.423, 65.424, 103.812, 105.845, 55.921, -153.967]
  MoveL 7046 to (-63.33, -8.94, -230.39) mm, rotated rx 81.04 ry 30.21 rz 20.91 deg; joints [-4.372, -5.363, 65.456, 103.81, 105.853, 55.825, -153.967]
  MoveL 7047 to (-64.3, -7.06, -230.41) mm, rotated rx 81.04 ry 30.21 rz 20.91 deg; joints [-4.342, -5.312, 65.5, 103.808, 105.862, 55.725, -153.967]
  MoveL 7048 to (-64.21, -6.43, -231.08) mm, rotated rx 81.04 ry 30.21 rz 20.91 deg; joints [-4.353, -5.257, 65.45, 103.798, 105.868, 55.721, -153.967]
  MoveL 7049 to (-63.99, -6.68, -231.41) mm, rotated rx 81.04 ry 30.21 rz 20.91 deg; joints [-4.363, -5.241, 65.406, 103.797, 105.866, 55.751, -153.967]
  MoveL 7050 to (-63.95, -6.71, -231.62) mm, rotated rx 81.04 ry 30.21 rz 20.91 deg; joints [-4.367, -5.226, 65.379, 103.797, 105.865, 55.763, -153.967]
  MoveL 7051 to (-64.09, -6.54, -231.72) mm, rotated rx 81.04 ry 30.21 rz 20.91 deg; joints [-4.364, -5.213, 65.368, 103.799, 105.864, 55.761, -153.967]
  MoveL 7052 to (-64.41, -6.26, -231.74) mm, rotated rx 81.04 ry 30.21 rz 20.91 deg; joints [-4.354, -5.199, 65.363, 103.805, 105.862, 55.75, -153.967]
  MoveC 7053 to (-65.27, -5.72, -231.74) mm, rotated rx 81.04 ry 30.21 rz 20.91 deg; joints [-4.328, -5.168, 65.349, 103.822, 105.853, 55.73, -153.967] to (-66.16, -5.23, -231.74) mm, rotated rx 81.04 ry 30.21 rz 20.91 deg; joints [-4.3, -5.137, 65.33, 103.842, 105.843, 55.714, -153.967]
  MoveL 7054 to (-66.16, -5.23, -231.74) mm, rotated rx 81.04 ry 30.21 rz 20.91 deg; joints [-4.3, -5.136, 65.33, 103.842, 105.843, 55.714, -153.967]
  MoveL 7055 to (-66.63, -4.96, -231.77) mm, rotated rx 81.04 ry 30.21 rz 20.91 deg; joints [-4.286, -5.118, 65.318, 103.852, 105.837, 55.706, -153.967]
  MoveL 7056 to (-67.09, -4.67, -231.81) mm, rotated rx 81.04 ry 30.21 rz 20.91 deg; joints [-4.272, -5.098, 65.303, 103.862, 105.832, 55.699, -153.967]
  MoveL 7057 to (-67.58, -4.36, -231.88) mm, rotated rx 81.04 ry 30.21 rz 20.91 deg; joints [-4.258, -5.075, 65.286, 103.872, 105.827, 55.691, -153.967]
  MoveL 7058 to (-68.08, -4.05, -231.92) mm, rotated rx 81.04 ry 30.21 rz 20.91 deg; joints [-4.243, -5.054, 65.272, 103.883, 105.821, 55.682, -153.967]
  MoveL 7059 to (-69.14, -3.45, -231.95) mm, rotated rx 81.04 ry 30.21 rz 20.91 deg; joints [-4.21, -5.015, 65.248, 103.906, 105.809, 55.663, -153.967]
  MoveL 7060 to (-69.62, -3.16, -231.98) mm, rotated rx 81.04 ry 30.21 rz 20.91 deg; joints [-4.196, -4.995, 65.234, 103.916, 105.803, 55.655, -153.967]
  MoveL 7061 to (-70.01, -2.89, -232.05) mm, rotated rx 81.04 ry 30.21 rz 20.91 deg; joints [-4.185, -4.975, 65.219, 103.924, 105.799, 55.649, -153.967]
  MoveL 7062 to (-70.36, -2.63, -232.14) mm, rotated rx 81.04 ry 30.21 rz 20.91 deg; joints [-4.175, -4.955, 65.203, 103.931, 105.795, 55.644, -153.967]
  MoveL 7063 to (-70.71, -2.4, -232.21) mm, rotated rx 81.04 ry 30.21 rz 20.91 deg; joints [-4.165, -4.938, 65.19, 103.938, 105.791, 55.638, -153.967]
  MoveL 7064 to (-71.1, -2.16, -232.24) mm, rotated rx 81.04 ry 30.21 rz 20.91 deg; joints [-4.153, -4.921, 65.178, 103.947, 105.787, 55.632, -153.967]
  MoveL 7065 to (-73.39, -0.9, -232.24) mm, rotated rx 81.04 ry 30.21 rz 20.91 deg; joints [-4.082, -4.84, 65.128, 103.998, 105.76, 55.592, -153.967]
  MoveL 7066 to (-75.8, 0.73, -232.59) mm, rotated rx 81.04 ry 30.21 rz 20.91 deg; joints [-4.012, -4.725, 65.045, 104.048, 105.734, 55.551, -153.967]
  MoveL 7067 to (-76.72, 1.62, -233.02) mm, rotated rx 81.04 ry 30.21 rz 20.91 deg; joints [-3.988, -4.655, 64.987, 104.064, 105.726, 55.535, -153.967]
  MoveL 7068 to (-77.46, 2.56, -233.62) mm, rotated rx 81.04 ry 30.21 rz 20.91 deg; joints [-3.973, -4.577, 64.919, 104.074, 105.721, 55.523, -153.967]
  MoveL 7069 to (-78, 3.56, -234.4) mm, rotated rx 81.04 ry 30.21 rz 20.91 deg; joints [-3.965, -4.49, 64.84, 104.078, 105.719, 55.515, -153.967]
  MoveL 7070 to (-78.36, 4.61, -235.35) mm, rotated rx 81.04 ry 30.21 rz 20.91 deg; joints [-3.965, -4.394, 64.75, 104.077, 105.72, 55.509, -153.967]
  MoveL 7071 to (-78.51, 6.86, -237.76) mm, rotated rx 81.04 ry 30.21 rz 20.91 deg; joints [-3.989, -4.178, 64.536, 104.056, 105.733, 55.51, -153.967]
  MoveL 7072 to (-77.99, 8.7, -240.17) mm, rotated rx 81.04 ry 30.21 rz 20.91 deg; joints [-4.034, -3.986, 64.334, 104.022, 105.752, 55.526, -153.967]
  MoveL 7073 to (-77.51, 9.22, -241.12) mm, rotated rx 81.04 ry 30.21 rz 20.91 deg; joints [-4.06, -3.921, 64.258, 104.003, 105.761, 55.539, -153.967]
  MoveL 7074 to (-76.88, 9.47, -241.9) mm, rotated rx 81.04 ry 30.21 rz 20.91 deg; joints [-4.088, -3.877, 64.2, 103.983, 105.772, 55.557, -153.967]
  MoveL 7075 to (-76.51, 9.5, -242.22) mm, rotated rx 81.04 ry 30.21 rz 20.91 deg; joints [-4.104, -3.862, 64.177, 103.972, 105.777, 55.568, -153.967]
  MoveL 7076 to (-76.11, 9.47, -242.5) mm, rotated rx 81.04 ry 30.21 rz 20.91 deg; joints [-4.119, -3.853, 64.158, 103.962, 105.782, 55.579, -153.967]
  MoveL 7077 to (-75.18, 9.2, -242.93) mm, rotated rx 81.04 ry 30.21 rz 20.91 deg; joints [-4.153, -3.85, 64.134, 103.939, 105.794, 55.604, -153.967]
  MoveL 7078 to (-74.12, 8.67, -243.19) mm, rotated rx 81.04 ry 30.21 rz 20.91 deg; joints [-4.189, -3.868, 64.127, 103.916, 105.805, 55.634, -153.967]
  MoveL 7079 to (-72.9, 7.88, -243.28) mm, rotated rx 81.04 ry 30.21 rz 20.91 deg; joints [-4.228, -3.906, 64.137, 103.892, 105.817, 55.667, -153.967]
  MoveL 7080 to (-72.47, 7.57, -243.28) mm, rotated rx 81.04 ry 30.21 rz 20.91 deg; joints [-4.241, -3.922, 64.143, 103.883, 105.821, 55.678, -153.967]
  MoveL 7081 to (-72.12, 7.29, -243.24) mm, rotated rx 81.04 ry 30.21 rz 20.91 deg; joints [-4.251, -3.938, 64.152, 103.877, 105.824, 55.688, -153.967]
  MoveL 7082 to (-71.8, 7.02, -243.19) mm, rotated rx 81.04 ry 30.21 rz 20.91 deg; joints [-4.26, -3.954, 64.161, 103.871, 105.827, 55.696, -153.967]
  MoveL 7083 to (-71.5, 6.75, -243.12) mm, rotated rx 81.04 ry 30.21 rz 20.91 deg; joints [-4.269, -3.972, 64.172, 103.866, 105.829, 55.703, -153.967]
  MoveL 7084 to (-71.16, 6.47, -243.07) mm, rotated rx 81.04 ry 30.21 rz 20.91 deg; joints [-4.279, -3.989, 64.181, 103.859, 105.832, 55.712, -153.967]
  MoveL 7085 to (-70.75, 6.16, -243.05) mm, rotated rx 81.04 ry 30.21 rz 20.91 deg; joints [-4.291, -4.006, 64.189, 103.852, 105.836, 55.723, -153.967]
  MoveL 7086 to (-66.1, 2.82, -243.04) mm, rotated rx 81.04 ry 30.21 rz 20.91 deg; joints [-4.435, -4.18, 64.254, 103.762, 105.879, 55.851, -153.967]
  MoveL 7087 to (-65.49, 2.36, -243.03) mm, rotated rx 81.04 ry 30.21 rz 20.91 deg; joints [-4.453, -4.204, 64.263, 103.751, 105.885, 55.869, -153.967]
  MoveL 7088 to (-64.98, 1.94, -243.02) mm, rotated rx 81.04 ry 30.21 rz 20.91 deg; joints [-4.469, -4.224, 64.268, 103.742, 105.889, 55.886, -153.967]
  MoveL 7089 to (-64.59, 1.52, -243.01) mm, rotated rx 81.04 ry 30.21 rz 20.91 deg; joints [-4.481, -4.241, 64.268, 103.737, 105.89, 55.905, -153.967]
  MoveL 7090 to (-64.29, 1.07, -242.97) mm, rotated rx 81.04 ry 30.21 rz 20.91 deg; joints [-4.49, -4.258, 64.266, 103.735, 105.89, 55.925, -153.967]
  MoveL 7091 to (-64.15, 0.77, -242.81) mm, rotated rx 81.04 ry 30.21 rz 20.91 deg; joints [-4.492, -4.278, 64.278, 103.735, 105.889, 55.933, -153.967]
  MoveL 7092 to (-64.18, 0.76, -242.5) mm, rotated rx 81.04 ry 30.21 rz 20.91 deg; joints [-4.487, -4.301, 64.318, 103.734, 105.891, 55.916, -153.967]
  MoveL 7093 to (-64.37, 1.07, -242.01) mm, rotated rx 81.04 ry 30.21 rz 20.91 deg; joints [-4.476, -4.329, 64.388, 103.732, 105.895, 55.872, -153.967]
  MoveL 7094 to (-64.76, 0.57, -241.04) mm, rotated rx 81.04 ry 30.21 rz 20.91 deg; joints [-4.453, -4.399, 64.472, 103.748, 105.888, 55.854, -153.967]
  MoveL 7095 to (-64.15, -1.19, -240.74) mm, rotated rx 81.04 ry 30.21 rz 20.91 deg; joints [-4.468, -4.46, 64.454, 103.757, 105.876, 55.936, -153.967]
  MoveL 7096 to (-63.49, -3.04, -240.53) mm, rotated rx 81.04 ry 30.21 rz 20.91 deg; joints [-4.485, -4.516, 64.421, 103.767, 105.864, 56.028, -153.967]
  MoveL 7097 to (-62.76, -5.04, -240.41) mm, rotated rx 81.04 ry 30.21 rz 20.91 deg; joints [-4.506, -4.569, 64.373, 103.778, 105.849, 56.133, -153.967]
  MoveL 7098 to (-61.27, -9.04, -240.41) mm, rotated rx 81.04 ry 30.21 rz 20.91 deg; joints [-4.551, -4.656, 64.243, 103.8, 105.82, 56.357, -153.967]
  MoveL 7099 to (-60.58, -10.9, -240.32) mm, rotated rx 81.04 ry 30.21 rz 20.91 deg; joints [-4.571, -4.703, 64.194, 103.81, 105.807, 56.457, -153.967]
  MoveL 7100 to (-59.83, -12.89, -240.32) mm, rotated rx 81.04 ry 30.21 rz 20.91 deg; joints [-4.593, -4.746, 64.129, 103.821, 105.792, 56.569, -153.967]
  MoveL 7101 to (-59.17, -14.95, -240.32) mm, rotated rx 81.04 ry 30.21 rz 20.91 deg; joints [-4.613, -4.787, 64.055, 103.836, 105.775, 56.687, -153.967]
  MoveL 7102 to (-58.42, -17.38, -240.14) mm, rotated rx 81.04 ry 30.21 rz 20.91 deg; joints [-4.634, -4.848, 63.99, 103.854, 105.754, 56.817, -153.967]
  MoveL 7103 to (-57.52, -19.42, -239.91) mm, rotated rx 81.04 ry 30.21 rz 20.91 deg; joints [-4.658, -4.913, 63.958, 103.86, 105.744, 56.917, -153.967]
  MoveL 7104 to (-56.67, -21.42, -239.79) mm, rotated rx 81.04 ry 30.21 rz 20.91 deg; joints [-4.682, -4.967, 63.911, 103.868, 105.732, 57.022, -153.967]
  MoveL 7105 to (-55.92, -23.42, -239.68) mm, rotated rx 81.04 ry 30.21 rz 20.91 deg; joints [-4.704, -5.017, 63.858, 103.879, 105.717, 57.13, -153.967]
  MoveL 7106 to (-55.17, -25.41, -239.47) mm, rotated rx 81.04 ry 30.21 rz 20.91 deg; joints [-4.724, -5.075, 63.818, 103.889, 105.704, 57.231, -153.967]
  MoveL 7107 to (-54.42, -27.41, -239.36) mm, rotated rx 81.04 ry 30.21 rz 20.91 deg; joints [-4.745, -5.124, 63.763, 103.9, 105.69, 57.339, -153.967]
  MoveL 7108 to (-53.66, -29.4, -239.25) mm, rotated rx 81.04 ry 30.21 rz 20.91 deg; joints [-4.766, -5.174, 63.708, 103.911, 105.675, 57.447, -153.967]
  MoveL 7109 to (-52.89, -31.39, -239.04) mm, rotated rx 81.04 ry 30.21 rz 20.91 deg; joints [-4.787, -5.231, 63.667, 103.921, 105.662, 57.548, -153.967]
  MoveL 7110 to (-52.13, -33.39, -238.93) mm, rotated rx 81.04 ry 30.21 rz 20.91 deg; joints [-4.808, -5.28, 63.611, 103.932, 105.648, 57.657, -153.967]
  MoveL 7111 to (-51.37, -35.38, -238.83) mm, rotated rx 81.04 ry 30.21 rz 20.91 deg; joints [-4.83, -5.328, 63.555, 103.943, 105.634, 57.765, -153.967]
  MoveL 7112 to (-50.59, -37.37, -238.62) mm, rotated rx 81.04 ry 30.21 rz 20.91 deg; joints [-4.851, -5.385, 63.513, 103.953, 105.621, 57.867, -153.967]
  MoveL 7113 to (-49.83, -39.36, -238.52) mm, rotated rx 81.04 ry 30.21 rz 20.91 deg; joints [-4.872, -5.432, 63.456, 103.964, 105.606, 57.976, -153.967]
  MoveL 7114 to (-49.09, -41.06, -238.26) mm, rotated rx 81.04 ry 30.21 rz 20.91 deg; joints [-4.891, -5.489, 63.433, 103.97, 105.597, 58.058, -153.967]
  MoveL 7115 to (-48.38, -42.57, -237.89) mm, rotated rx 81.04 ry 30.21 rz 20.91 deg; joints [-4.908, -5.551, 63.433, 103.972, 105.591, 58.122, -153.967]
  MoveL 7116 to (-47.66, -43.91, -237.39) mm, rotated rx 81.04 ry 30.21 rz 20.91 deg; joints [-4.924, -5.622, 63.461, 103.971, 105.589, 58.169, -153.967]
  MoveL 7117 to (-47.81, -42.79, -236.55) mm, rotated rx 81.04 ry 30.21 rz 20.91 deg; joints [-4.911, -5.674, 63.627, 103.952, 105.609, 58.052, -153.967]
  MoveL 7118 to (-47.7, -43.1, -236.52) mm, rotated rx 81.04 ry 30.21 rz 20.91 deg; joints [-4.914, -5.682, 63.619, 103.954, 105.607, 58.068, -153.967]
  MoveL 7119 to (-47.62, -43.41, -236.48) mm, rotated rx 81.04 ry 30.21 rz 20.91 deg; joints [-4.915, -5.691, 63.612, 103.956, 105.604, 58.085, -153.967]
  MoveL 7120 to (-47.61, -43.78, -236.42) mm, rotated rx 81.04 ry 30.21 rz 20.91 deg; joints [-4.915, -5.699, 63.599, 103.962, 105.599, 58.105, -153.967]
  MoveL 7121 to (-47.64, -44.19, -236.39) mm, rotated rx 81.04 ry 30.21 rz 20.91 deg; joints [-4.913, -5.704, 63.58, 103.97, 105.592, 58.13, -153.967]
  MoveL 7122 to (-47.73, -44.67, -236.36) mm, rotated rx 81.04 ry 30.21 rz 20.91 deg; joints [-4.91, -5.708, 63.553, 103.981, 105.583, 58.16, -153.967]
  MoveL 7123 to (-48.81, -49.26, -236.36) mm, rotated rx 81.04 ry 30.21 rz 20.91 deg; joints [-4.875, -5.715, 63.248, 104.093, 105.489, 58.469, -153.967]
  MoveL 7124 to (-48.89, -49.65, -236.33) mm, rotated rx 81.04 ry 30.21 rz 20.91 deg; joints [-4.873, -5.718, 63.227, 104.102, 105.482, 58.494, -153.967]
  MoveL 7125 to (-49.01, -50.16, -236.33) mm, rotated rx 81.04 ry 30.21 rz 20.91 deg; joints [-4.869, -5.718, 63.192, 104.115, 105.471, 58.528, -153.967]
  MoveL 7126 to (-49.22, -51.17, -236.3) mm, rotated rx 81.04 ry 30.21 rz 20.91 deg; joints [-4.861, -5.723, 63.131, 104.138, 105.451, 58.594, -153.967]
  MoveL 7127 to (-49.82, -53.72, -236.3) mm, rotated rx 81.04 ry 30.21 rz 20.91 deg; joints [-4.842, -5.726, 62.96, 104.2, 105.399, 58.766, -153.967]
  MoveL 7128 to (-50, -54.73, -236.28) mm, rotated rx 81.04 ry 30.21 rz 20.91 deg; joints [-4.836, -5.729, 62.896, 104.223, 105.379, 58.833, -153.967]
  MoveL 7129 to (-50.32, -56.14, -236.34) mm, rotated rx 81.04 ry 30.21 rz 20.91 deg; joints [-4.827, -5.726, 62.793, 104.257, 105.349, 58.932, -153.967]
  MoveL 7130 to (-50.71, -57.25, -236.6) mm, rotated rx 81.04 ry 30.21 rz 20.91 deg; joints [-4.817, -5.702, 62.677, 104.29, 105.322, 59.023, -153.967]
  MoveL 7131 to (-51.19, -58.05, -237.04) mm, rotated rx 81.04 ry 30.21 rz 20.91 deg; joints [-4.807, -5.659, 62.55, 104.32, 105.296, 59.107, -153.967]
  MoveL 7132 to (-51.45, -58.33, -237.33) mm, rotated rx 81.04 ry 30.21 rz 20.91 deg; joints [-4.802, -5.631, 62.481, 104.334, 105.283, 59.146, -153.967]
  MoveL 7133 to (-51.74, -58.54, -237.66) mm, rotated rx 81.04 ry 30.21 rz 20.91 deg; joints [-4.797, -5.597, 62.41, 104.348, 105.271, 59.183, -153.967]
  MoveL 7134 to (-52.37, -58.73, -238.48) mm, rotated rx 81.04 ry 30.21 rz 20.91 deg; joints [-4.787, -5.515, 62.259, 104.375, 105.249, 59.251, -153.967]
  MoveL 7135 to (-53.07, -58.61, -239.47) mm, rotated rx 81.04 ry 30.21 rz 20.91 deg; joints [-4.777, -5.414, 62.096, 104.399, 105.228, 59.312, -153.967]
  MoveL 7136 to (-54.73, -57.46, -242.03) mm, rotated rx 81.04 ry 30.21 rz 20.91 deg; joints [-4.756, -5.152, 61.732, 104.443, 105.191, 59.411, -153.967]
  MoveL 7137 to (-56.17, -55.55, -244.6) mm, rotated rx 81.04 ry 30.21 rz 20.91 deg; joints [-4.741, -4.89, 61.419, 104.468, 105.171, 59.46, -153.967]
  MoveL 7138 to (-56.9, -53.33, -246.43) mm, rotated rx 81.04 ry 30.21 rz 20.91 deg; joints [-4.74, -4.705, 61.258, 104.462, 105.176, 59.436, -153.967]
  MoveL 7139 to (-56.99, -52.1, -247.07) mm, rotated rx 81.04 ry 30.21 rz 20.91 deg; joints [-4.745, -4.642, 61.235, 104.448, 105.189, 59.396, -153.967]
  MoveL 7140 to (-56.89, -50.8, -247.53) mm, rotated rx 81.04 ry 30.21 rz 20.91 deg; joints [-4.754, -4.599, 61.251, 104.426, 105.208, 59.338, -153.967]
  MoveL 7141 to (-56.16, -47.97, -247.89) mm, rotated rx 81.04 ry 30.21 rz 20.91 deg; joints [-4.781, -4.571, 61.398, 104.358, 105.266, 59.166, -153.967]
  MoveL 7142 to (-55.09, -45.02, -247.89) mm, rotated rx 81.04 ry 30.21 rz 20.91 deg; joints [-4.815, -4.581, 61.619, 104.275, 105.336, 58.96, -153.967]
  MoveL 7143 to (-54.76, -44.06, -247.91) mm, rotated rx 81.04 ry 30.21 rz 20.91 deg; joints [-4.825, -4.582, 61.687, 104.248, 105.358, 58.894, -153.967]
  MoveL 7144 to (-54.4, -43.08, -247.91) mm, rotated rx 81.04 ry 30.21 rz 20.91 deg; joints [-4.836, -4.585, 61.76, 104.221, 105.381, 58.825, -153.967]
  MoveL 7145 to (-54.23, -42.61, -247.91) mm, rotated rx 81.04 ry 30.21 rz 20.91 deg; joints [-4.842, -4.586, 61.794, 104.208, 105.392, 58.793, -153.967]
  MoveL 7146 to (-54.02, -41.98, -247.94) mm, rotated rx 81.04 ry 30.21 rz 20.91 deg; joints [-4.849, -4.585, 61.835, 104.191, 105.406, 58.751, -153.967]
  MoveL 7147 to (-53.84, -41.41, -248) mm, rotated rx 81.04 ry 30.21 rz 20.91 deg; joints [-4.855, -4.582, 61.869, 104.176, 105.418, 58.715, -153.967]
  MoveL 7148 to (-53.71, -40.92, -248.07) mm, rotated rx 81.04 ry 30.21 rz 20.91 deg; joints [-4.86, -4.576, 61.892, 104.164, 105.428, 58.686, -153.967]
  MoveL 7149 to (-53.58, -40.48, -248.12) mm, rotated rx 81.04 ry 30.21 rz 20.91 deg; joints [-4.865, -4.572, 61.916, 104.153, 105.438, 58.659, -153.967]
  MoveL 7150 to (-53.44, -40.03, -248.16) mm, rotated rx 81.04 ry 30.21 rz 20.91 deg; joints [-4.87, -4.57, 61.943, 104.141, 105.447, 58.63, -153.967]
  MoveL 7151 to (-52.9, -38.56, -248.16) mm, rotated rx 81.04 ry 30.21 rz 20.91 deg; joints [-4.887, -4.574, 62.051, 104.099, 105.481, 58.527, -153.967]
  MoveL 7152 to (-52.75, -38.08, -248.17) mm, rotated rx 81.04 ry 30.21 rz 20.91 deg; joints [-4.892, -4.573, 62.083, 104.086, 105.492, 58.495, -153.967]
  MoveL 7153 to (-52.63, -37.65, -248.2) mm, rotated rx 81.04 ry 30.21 rz 20.91 deg; joints [-4.896, -4.571, 62.109, 104.076, 105.501, 58.468, -153.967]
  MoveL 7154 to (-52.57, -37.27, -248.24) mm, rotated rx 81.04 ry 30.21 rz 20.91 deg; joints [-4.898, -4.566, 62.127, 104.067, 105.508, 58.445, -153.967]
  MoveL 7155 to (-52.57, -36.97, -248.31) mm, rotated rx 81.04 ry 30.21 rz 20.91 deg; joints [-4.899, -4.558, 62.134, 104.063, 105.512, 58.43, -153.967]
  MoveL 7156 to (-52.62, -36.7, -248.38) mm, rotated rx 81.04 ry 30.21 rz 20.91 deg; joints [-4.898, -4.549, 62.137, 104.06, 105.514, 58.418, -153.967]
  MoveL 7157 to (-52.94, -38.26, -249.18) mm, rotated rx 81.04 ry 30.21 rz 20.91 deg; joints [-4.897, -4.488, 61.925, 104.102, 105.477, 58.569, -153.967]
  MoveL 7158 to (-53.33, -36.53, -249.59) mm, rotated rx 81.04 ry 30.21 rz 20.91 deg; joints [-4.89, -4.43, 61.947, 104.086, 105.493, 58.489, -153.967]
  MoveL 7159 to (-53.76, -34.71, -249.85) mm, rotated rx 81.04 ry 30.21 rz 20.91 deg; joints [-4.881, -4.381, 61.989, 104.069, 105.51, 58.395, -153.967]
  MoveL 7160 to (-54.25, -32.77, -250.03) mm, rotated rx 81.04 ry 30.21 rz 20.91 deg; joints [-4.869, -4.336, 62.046, 104.051, 105.529, 58.291, -153.967]
  MoveL 7161 to (-54.79, -30.7, -250.23) mm, rotated rx 81.04 ry 30.21 rz 20.91 deg; joints [-4.855, -4.287, 62.106, 104.033, 105.548, 58.18, -153.967]
  MoveL 7162 to (-55.31, -28.63, -250.32) mm, rotated rx 81.04 ry 30.21 rz 20.91 deg; joints [-4.841, -4.246, 62.179, 104.013, 105.568, 58.063, -153.967]
  MoveL 7163 to (-55.83, -26.56, -250.42) mm, rotated rx 81.04 ry 30.21 rz 20.91 deg; joints [-4.827, -4.205, 62.252, 103.994, 105.589, 57.946, -153.967]
  MoveL 7164 to (-56.36, -24.5, -250.62) mm, rotated rx 81.04 ry 30.21 rz 20.91 deg; joints [-4.814, -4.155, 62.31, 103.976, 105.608, 57.835, -153.967]
  MoveL 7165 to (-56.87, -22.42, -250.72) mm, rotated rx 81.04 ry 30.21 rz 20.91 deg; joints [-4.8, -4.113, 62.382, 103.956, 105.628, 57.719, -153.967]
  MoveL 7166 to (-57.39, -20.35, -250.82) mm, rotated rx 81.04 ry 30.21 rz 20.91 deg; joints [-4.786, -4.07, 62.453, 103.937, 105.649, 57.603, -153.967]
  MoveL 7167 to (-57.9, -18.28, -251.02) mm, rotated rx 81.04 ry 30.21 rz 20.91 deg; joints [-4.773, -4.02, 62.509, 103.918, 105.668, 57.493, -153.967]
  MoveL 7168 to (-58.92, -14.14, -251.22) mm, rotated rx 81.04 ry 30.21 rz 20.91 deg; joints [-4.745, -3.934, 62.65, 103.879, 105.708, 57.261, -153.967]
  MoveL 7169 to (-59.35, -12.4, -251.43) mm, rotated rx 81.04 ry 30.21 rz 20.91 deg; joints [-4.735, -3.887, 62.691, 103.863, 105.724, 57.171, -153.967]
  MoveL 7170 to (-59.85, -10.5, -251.5) mm, rotated rx 81.04 ry 30.21 rz 20.91 deg; joints [-4.721, -3.848, 62.755, 103.846, 105.742, 57.065, -153.967]
  MoveL 7171 to (-60.43, -8.53, -251.51) mm, rotated rx 81.04 ry 30.21 rz 20.91 deg; joints [-4.704, -3.81, 62.827, 103.83, 105.76, 56.952, -153.967]
  MoveL 7172 to (-61.05, -5.93, -251.62) mm, rotated rx 81.04 ry 30.21 rz 20.91 deg; joints [-4.687, -3.756, 62.915, 103.806, 105.785, 56.807, -153.967]
  MoveL 7173 to (-61.54, -3.4, -251.71) mm, rotated rx 81.04 ry 30.21 rz 20.91 deg; joints [-4.673, -3.707, 63.007, 103.778, 105.812, 56.663, -153.967]
  MoveL 7174 to (-62.02, -1.24, -251.81) mm, rotated rx 81.04 ry 30.21 rz 20.91 deg; joints [-4.661, -3.663, 63.08, 103.756, 105.834, 56.542, -153.967]
  MoveL 7175 to (-62.49, 0.75, -251.98) mm, rotated rx 81.04 ry 30.21 rz 20.91 deg; joints [-4.649, -3.614, 63.135, 103.737, 105.852, 56.436, -153.967]
  MoveL 7176 to (-62.91, 2.61, -252.26) mm, rotated rx 81.04 ry 30.21 rz 20.91 deg; joints [-4.639, -3.559, 63.17, 103.72, 105.869, 56.345, -153.967]
  MoveL 7177 to (-63.32, 4.46, -252.55) mm, rotated rx 81.04 ry 30.21 rz 20.91 deg; joints [-4.631, -3.504, 63.204, 103.703, 105.886, 56.254, -153.967]
  MoveL 7178 to (-63.69, 6.3, -252.84) mm, rotated rx 81.04 ry 30.21 rz 20.91 deg; joints [-4.623, -3.449, 63.238, 103.685, 105.903, 56.163, -153.967]
  MoveL 7179 to (-64.13, 8.24, -253) mm, rotated rx 81.04 ry 30.21 rz 20.91 deg; joints [-4.612, -3.402, 63.291, 103.666, 105.921, 56.06, -153.967]
  MoveL 7180 to (-63.79, 8.81, -253.62) mm, rotated rx 81.04 ry 30.21 rz 20.91 deg; joints [-4.629, -3.357, 63.252, 103.65, 105.931, 56.056, -153.967]
  MoveL 7181 to (-63.59, 8.56, -253.93) mm, rotated rx 81.04 ry 30.21 rz 20.91 deg; joints [-4.639, -3.342, 63.208, 103.65, 105.93, 56.086, -153.967]
  MoveL 7182 to (-63.54, 8.57, -254.12) mm, rotated rx 81.04 ry 30.21 rz 20.91 deg; joints [-4.643, -3.328, 63.185, 103.649, 105.929, 56.096, -153.967]
  MoveL 7183 to (-63.65, 8.79, -254.22) mm, rotated rx 81.04 ry 30.21 rz 20.91 deg; joints [-4.641, -3.314, 63.178, 103.649, 105.929, 56.09, -153.967]
  MoveL 7184 to (-63.92, 9.15, -254.24) mm, rotated rx 81.04 ry 30.21 rz 20.91 deg; joints [-4.633, -3.301, 63.18, 103.652, 105.929, 56.073, -153.967]
  MoveL 7185 to (-64.24, 9.52, -254.24) mm, rotated rx 81.04 ry 30.21 rz 20.91 deg; joints [-4.623, -3.287, 63.181, 103.655, 105.928, 56.056, -153.967]
  MoveL 7186 to (-64.96, 10.18, -254.27) mm, rotated rx 81.04 ry 30.21 rz 20.91 deg; joints [-4.601, -3.256, 63.174, 103.667, 105.923, 56.029, -153.967]
  MoveL 7187 to (-66.12, 11.24, -254.27) mm, rotated rx 81.04 ry 30.21 rz 20.91 deg; joints [-4.566, -3.21, 63.169, 103.685, 105.916, 55.984, -153.967]
  MoveL 7188 to (-66.81, 11.93, -254.29) mm, rotated rx 81.04 ry 30.21 rz 20.91 deg; joints [-4.544, -3.18, 63.166, 103.696, 105.911, 55.954, -153.967]
  MoveL 7189 to (-67.59, 12.64, -254.29) mm, rotated rx 81.04 ry 30.21 rz 20.91 deg; joints [-4.521, -3.15, 63.162, 103.708, 105.906, 55.924, -153.967]
  MoveL 7190 to (-67.96, 12.99, -254.3) mm, rotated rx 81.04 ry 30.21 rz 20.91 deg; joints [-4.509, -3.133, 63.159, 103.714, 105.904, 55.91, -153.967]
  MoveL 7191 to (-68.3, 13.32, -254.33) mm, rotated rx 81.04 ry 30.21 rz 20.91 deg; joints [-4.499, -3.117, 63.154, 103.719, 105.902, 55.897, -153.967]
  MoveL 7192 to (-68.61, 13.63, -254.38) mm, rotated rx 81.04 ry 30.21 rz 20.91 deg; joints [-4.49, -3.101, 63.148, 103.724, 105.9, 55.886, -153.967]
